DATA_BLOCK "DB240_Program10"   // DB240
{ S7_Optimized_Access := 'FALSE' }
AUTHOR : Robopac
VERSION : 0.0
// stored: AutoNumber false, IsOnlyStoredInLoadMemory false, IsWriteProtectedInAS false
   VAR RETAIN
      Program10 { S7_SetPoint := 'True'} : "DatiProgramma";
   END_VAR
BEGIN
   Program10.Wrapping := TRUE;
   Program10.TopLenght := 500;
   Program10.TopRelease := 0;
   Program10.TopDown := 0;
   Program10.Top := 4;
   Program10.PressurePTime := 0;
   Program10.LifterTime := 0;
   Program10.RevOverContrast := 1;
   Program10.RopeEndCycle := 16#02;
   Program10.Spare4 := 16#01;
   Program10.RopeTime := 1500;
   Program10.RevOverClamp := 1;
   Program10.FilmForceFinalRev := 10;
   Program10.FilmPrestretchFinalRev := 100;
   Program10.ArmSpeed := 100;
   Program10.CarriageDown4Top := 500;
   Program10.TopDownTime := 1500;
   Program10.LapsUnderTop := 0;
   Program10.Spare6 := 0;
   Program10.Spare7 := 0;
   Program10.Spare8 := 0;
   Program10.Spare9 := 0;
   Program10.Spare10 := 0;
   Program10.Spare11 := 0;
   Program10.Spare12 := 0;
   Program10.Overlap0_1 := 0;
   Program10.Height1 := 130;
   Program10.Landmark1 := FALSE;
   Program10.Lifter1 := FALSE;
   Program10.SpareBit1H1 := FALSE;
   Program10.Airblower1 := TRUE;
   Program10.NextStep1 := TRUE;
   Program10.PressureP1 := TRUE;
   Program10.SpareByte2H1 := 16#00;
   Program10.Revolution1 := 1;
   Program10.RopeUnit1_1 := 16#01;
   Program10.RopeUnit1_2 := 16#01;
   Program10.FilmForce1 := 5;
   Program10.FilmPrestretch1 := 200;
   Program10.Spare3H1 := 0;
   Program10.Spare49 := 0;
   Program10.Spare50 := 0;
   Program10.Spare51 := 0;
   Program10.Spare52 := 0;
   Program10.Spare53 := 0;
   Program10.Overlap1_2 := 0;
   Program10.Height2 := 50;
   Program10.Landmark2 := FALSE;
   Program10.Lifter2 := FALSE;
   Program10.SpareBit1H2 := FALSE;
   Program10.Airblower2 := TRUE;
   Program10.NextStep2 := TRUE;
   Program10.PressureP2 := TRUE;
   Program10.SpareByte2H2 := 16#00;
   Program10.Revolution2 := 1;
   Program10.RopeUnit2_1 := 16#01;
   Program10.RopeUnit2_2 := 16#01;
   Program10.FilmForce2 := 20;
   Program10.FilmPrestretch2 := 200;
   Program10.Spare3H2 := 0;
   Program10.Spare54 := 0;
   Program10.Spare55 := 0;
   Program10.Spare56 := 0;
   Program10.Spare57 := 0;
   Program10.Spare58 := 0;
   Program10.Overlap2_3 := 100;
   Program10.Height3 := -50;
   Program10.Landmark3 := TRUE;
   Program10.Lifter3 := FALSE;
   Program10.SpareBit1H3 := FALSE;
   Program10.Airblower3 := TRUE;
   Program10.NextStep3 := TRUE;
   Program10.PressureP3 := TRUE;
   Program10.SpareByte2H3 := 16#00;
   Program10.Revolution3 := 2;
   Program10.RopeUnit3_1 := 16#01;
   Program10.RopeUnit3_2 := 16#01;
   Program10.FilmForce3 := 30;
   Program10.FilmPrestretch3 := 200;
   Program10.Spare3H3 := 0;
   Program10.Spare59 := 0;
   Program10.Spare60 := 0;
   Program10.Spare61 := 380;
   Program10.Spare62 := 2800;
   Program10.Spare63 := 0;
   Program10.Overlap3_4 := 100;
   Program10.Height4 := 100;
   Program10.Landmark4 := FALSE;
   Program10.Lifter4 := FALSE;
   Program10.SpareBit1H4 := FALSE;
   Program10.Airblower4 := TRUE;
   Program10.NextStep4 := TRUE;
   Program10.PressureP4 := TRUE;
   Program10.SpareByte2H4 := 16#00;
   Program10.Revolution4 := 3;
   Program10.RopeUnit4_1 := 16#02;
   Program10.RopeUnit4_2 := 16#02;
   Program10.FilmForce4 := 30;
   Program10.FilmPrestretch4 := 200;
   Program10.Spare3H4 := 0;
   Program10.Spare64 := 0;
   Program10.Spare65 := 0;
   Program10.Spare66 := 0;
   Program10.Spare67 := 0;
   Program10.Spare68 := 0;
   Program10.Overlap4_5 := 0;
   Program10.Height5 := 50;
   Program10.Landmark5 := FALSE;
   Program10.Lifter5 := FALSE;
   Program10.SpareBit1H5 := FALSE;
   Program10.Airblower5 := TRUE;
   Program10.NextStep5 := FALSE;
   Program10.PressureP5 := FALSE;
   Program10.SpareByte2H5 := 16#00;
   Program10.Revolution5 := 1;
   Program10.RopeUnit5_1 := 16#01;
   Program10.RopeUnit5_2 := 16#01;
   Program10.FilmForce5 := 30;
   Program10.FilmPrestretch5 := 200;
   Program10.Spare3H5 := 0;
   Program10.Spare69 := 0;
   Program10.Spare70 := 0;
   Program10.Spare71 := 0;
   Program10.Spare72 := 0;
   Program10.Spare73 := 0;
   Program10.Overlap5_6 := 100;
   Program10.Height6 := 50;
   Program10.Landmark6 := FALSE;
   Program10.Lifter6 := FALSE;
   Program10.SpareBit1H6 := FALSE;
   Program10.Airblower6 := TRUE;
   Program10.NextStep6 := FALSE;
   Program10.PressureP6 := FALSE;
   Program10.SpareByte2H6 := 16#00;
   Program10.Revolution6 := 2;
   Program10.RopeUnit6_1 := 16#02;
   Program10.RopeUnit6_2 := 16#01;
   Program10.FilmForce6 := 20;
   Program10.FilmPrestretch6 := 200;
   Program10.Spare3H6 := 0;
   Program10.Spare74 := 0;
   Program10.Spare75 := 0;
   Program10.Spare76 := 0;
   Program10.Spare77 := 0;
   Program10.Spare78 := 0;
   Program10.Overlap6_7 := 0;
   Program10.Height7 := 0;
   Program10.Landmark7 := FALSE;
   Program10.Lifter7 := FALSE;
   Program10.SpareBit1H7 := FALSE;
   Program10.Airblower7 := FALSE;
   Program10.NextStep7 := TRUE;
   Program10.PressureP7 := FALSE;
   Program10.SpareByte2H7 := 16#00;
   Program10.Revolution7 := 1;
   Program10.RopeUnit7_1 := 16#01;
   Program10.RopeUnit7_2 := 16#01;
   Program10.FilmForce7 := 0;
   Program10.FilmPrestretch7 := 100;
   Program10.Spare3H7 := 0;
   Program10.Spare79 := 0;
   Program10.Spare80 := 0;
   Program10.Spare81 := 0;
   Program10.Spare82 := 0;
   Program10.Spare83 := 0;
   Program10.Overlap7_8 := 0;
   Program10.Height8 := 0;
   Program10.Landmark8 := FALSE;
   Program10.Lifter8 := FALSE;
   Program10.SpareBit1H8 := FALSE;
   Program10.Airblower8 := FALSE;
   Program10.NextStep8 := TRUE;
   Program10.PressureP8 := FALSE;
   Program10.SpareByte2H8 := 16#00;
   Program10.Revolution8 := 1;
   Program10.RopeUnit8_1 := 16#01;
   Program10.RopeUnit8_2 := 16#01;
   Program10.FilmForce8 := 0;
   Program10.FilmPrestretch8 := 100;
   Program10.Spare3H8 := 0;
   Program10.Spare84 := 0;
   Program10.Spare85 := 0;
   Program10.Spare86 := 0;
   Program10.Spare87 := 0;
   Program10.Spare88 := 0;
   Program10.Overlap8_9 := 0;
   Program10.Height9 := 0;
   Program10.Landmark9 := FALSE;
   Program10.Lifter9 := FALSE;
   Program10.SpareBit1H9 := FALSE;
   Program10.Airblower9 := FALSE;
   Program10.NextStep9 := TRUE;
   Program10.PressureP9 := FALSE;
   Program10.SpareByte2H9 := 16#00;
   Program10.Revolution9 := 1;
   Program10.RopeUnit9_1 := 16#01;
   Program10.RopeUnit9_2 := 16#01;
   Program10.FilmForce9 := 0;
   Program10.FilmPrestretch9 := 100;
   Program10.Spare3H9 := 0;
   Program10.Spare89 := 0;
   Program10.Spare90 := 0;
   Program10.Spare91 := 0;
   Program10.Spare92 := 0;
   Program10.Spare93 := 0;
   Program10.Overlap9_10 := 0;
   Program10.Height10 := 0;
   Program10.Landmark10 := FALSE;
   Program10.Lifter10 := FALSE;
   Program10.SpareBit1H10 := FALSE;
   Program10.Airblower10 := FALSE;
   Program10.NextStep10 := FALSE;
   Program10.PressureP10 := FALSE;
   Program10.SpareByte2H10 := 16#00;
   Program10.Revolution10 := 1;
   Program10.RopeUnit10_1 := 16#01;
   Program10.RopeUnit10_2 := 16#01;
   Program10.FilmForce10 := 0;
   Program10.FilmPrestretch10 := 100;
   Program10.Spare3H10 := 0;
   Program10.Spare94 := 0;
   Program10.Spare95 := 0;
   Program10.Spare96 := 0;
   Program10.Spare97 := 0;
   Program10.Spare98 := 0;
   Program10.Overlap10_11 := 0;
   Program10.Height11 := 0;
   Program10.Landmark11 := FALSE;
   Program10.Lifter11 := FALSE;
   Program10.SpareBit1H11 := FALSE;
   Program10.Airblower11 := FALSE;
   Program10.NextStep11 := TRUE;
   Program10.PressureP11 := FALSE;
   Program10.SpareByte2H11 := 16#00;
   Program10.Revolution11 := 1;
   Program10.RopeUnit11_1 := 16#01;
   Program10.RopeUnit11_2 := 16#01;
   Program10.FilmForce11 := 0;
   Program10.FilmPrestretch11 := 100;
   Program10.Spare3H11 := 0;
   Program10.Spare99 := 0;
   Program10.Spare100 := 0;
   Program10.Spare101 := 0;
   Program10.Spare102 := 0;
   Program10.Spare103 := 0;
   Program10.Overlap11_12 := 0;
   Program10.Height12 := 0;
   Program10.Landmark12 := FALSE;
   Program10.Lifter12 := FALSE;
   Program10.SpareBit1H12 := FALSE;
   Program10.Airblower12 := FALSE;
   Program10.NextStep12 := FALSE;
   Program10.PressureP12 := FALSE;
   Program10.SpareByte2H12 := 16#00;
   Program10.Revolution12 := 1;
   Program10.RopeUnit12_1 := 16#01;
   Program10.RopeUnit12_2 := 16#01;
   Program10.FilmForce12 := 0;
   Program10.FilmPrestretch12 := 100;
   Program10.Spare3H12 := 0;
   Program10.Spare104 := 0;
   Program10.Spare105 := 0;
   Program10.Spare106 := 0;
   Program10.Spare107 := 0;
   Program10.Spare108 := 0;
END_DATA_BLOCK

DATA_BLOCK "DB243_Program7"   // DB243
{ S7_Optimized_Access := 'FALSE' }
AUTHOR : Robopac
VERSION : 0.0
// stored: AutoNumber false, IsOnlyStoredInLoadMemory false, IsWriteProtectedInAS false
   VAR RETAIN
      Program7 { S7_SetPoint := 'True'} : "DatiProgramma";
   END_VAR
BEGIN
   Program7.Wrapping := TRUE;
   Program7.TopLenght := 500;
   Program7.TopRelease := 0;
   Program7.TopDown := 0;
   Program7.Top := 4;
   Program7.PressurePTime := 0;
   Program7.LifterTime := 0;
   Program7.RevOverContrast := 1;
   Program7.RopeEndCycle := 16#01;
   Program7.Spare4 := 16#01;
   Program7.RopeTime := 1500;
   Program7.RevOverClamp := 1;
   Program7.FilmForceFinalRev := 15;
   Program7.FilmPrestretchFinalRev := 100;
   Program7.ArmSpeed := 100;
   Program7.CarriageDown4Top := 500;
   Program7.TopDownTime := 1500;
   Program7.LapsUnderTop := 0;
   Program7.Spare6 := 0;
   Program7.Spare7 := 0;
   Program7.Spare8 := 0;
   Program7.Spare9 := 0;
   Program7.Spare10 := 0;
   Program7.Spare11 := 0;
   Program7.Spare12 := 0;
   Program7.Overlap0_1 := 0;
   Program7.Height1 := 15;
   Program7.Landmark1 := FALSE;
   Program7.Lifter1 := FALSE;
   Program7.SpareBit1H1 := FALSE;
   Program7.Airblower1 := TRUE;
   Program7.NextStep1 := TRUE;
   Program7.PressureP1 := TRUE;
   Program7.SpareByte2H1 := 16#00;
   Program7.Revolution1 := 0;
   Program7.RopeUnit1_1 := 16#02;
   Program7.RopeUnit1_2 := 16#01;
   Program7.FilmForce1 := 5;
   Program7.FilmPrestretch1 := 200;
   Program7.Spare3H1 := 0;
   Program7.Spare49 := 0;
   Program7.Spare50 := 0;
   Program7.Spare51 := 0;
   Program7.Spare52 := 0;
   Program7.Spare53 := 0;
   Program7.Overlap1_2 := 0;
   Program7.Height2 := 80;
   Program7.Landmark2 := FALSE;
   Program7.Lifter2 := FALSE;
   Program7.SpareBit1H2 := FALSE;
   Program7.Airblower2 := TRUE;
   Program7.NextStep2 := TRUE;
   Program7.PressureP2 := TRUE;
   Program7.SpareByte2H2 := 16#00;
   Program7.Revolution2 := 1;
   Program7.RopeUnit2_1 := 16#01;
   Program7.RopeUnit2_2 := 16#01;
   Program7.FilmForce2 := 15;
   Program7.FilmPrestretch2 := 200;
   Program7.Spare3H2 := 0;
   Program7.Spare54 := 0;
   Program7.Spare55 := 0;
   Program7.Spare56 := 0;
   Program7.Spare57 := 0;
   Program7.Spare58 := 0;
   Program7.Overlap2_3 := 0;
   Program7.Height3 := 120;
   Program7.Landmark3 := FALSE;
   Program7.Lifter3 := FALSE;
   Program7.SpareBit1H3 := FALSE;
   Program7.Airblower3 := TRUE;
   Program7.NextStep3 := TRUE;
   Program7.PressureP3 := TRUE;
   Program7.SpareByte2H3 := 16#00;
   Program7.Revolution3 := 1;
   Program7.RopeUnit3_1 := 16#01;
   Program7.RopeUnit3_2 := 16#01;
   Program7.FilmForce3 := 25;
   Program7.FilmPrestretch3 := 200;
   Program7.Spare3H3 := 0;
   Program7.Spare59 := 0;
   Program7.Spare60 := 0;
   Program7.Spare61 := 380;
   Program7.Spare62 := 2800;
   Program7.Spare63 := 0;
   Program7.Overlap3_4 := 0;
   Program7.Height4 := -100;
   Program7.Landmark4 := TRUE;
   Program7.Lifter4 := FALSE;
   Program7.SpareBit1H4 := FALSE;
   Program7.Airblower4 := FALSE;
   Program7.NextStep4 := TRUE;
   Program7.PressureP4 := TRUE;
   Program7.SpareByte2H4 := 16#00;
   Program7.Revolution4 := 1;
   Program7.RopeUnit4_1 := 16#01;
   Program7.RopeUnit4_2 := 16#01;
   Program7.FilmForce4 := 20;
   Program7.FilmPrestretch4 := 200;
   Program7.Spare3H4 := 0;
   Program7.Spare64 := 0;
   Program7.Spare65 := 0;
   Program7.Spare66 := 0;
   Program7.Spare67 := 0;
   Program7.Spare68 := 0;
   Program7.Overlap4_5 := 300;
   Program7.Height5 := 120;
   Program7.Landmark5 := FALSE;
   Program7.Lifter5 := FALSE;
   Program7.SpareBit1H5 := FALSE;
   Program7.Airblower5 := TRUE;
   Program7.NextStep5 := TRUE;
   Program7.PressureP5 := FALSE;
   Program7.SpareByte2H5 := 16#00;
   Program7.Revolution5 := 2;
   Program7.RopeUnit5_1 := 16#02;
   Program7.RopeUnit5_2 := 16#02;
   Program7.FilmForce5 := 15;
   Program7.FilmPrestretch5 := 200;
   Program7.Spare3H5 := 0;
   Program7.Spare69 := 0;
   Program7.Spare70 := 0;
   Program7.Spare71 := 0;
   Program7.Spare72 := 0;
   Program7.Spare73 := 0;
   Program7.Overlap5_6 := 300;
   Program7.Height6 := 85;
   Program7.Landmark6 := FALSE;
   Program7.Lifter6 := FALSE;
   Program7.SpareBit1H6 := FALSE;
   Program7.Airblower6 := TRUE;
   Program7.NextStep6 := FALSE;
   Program7.PressureP6 := FALSE;
   Program7.SpareByte2H6 := 16#00;
   Program7.Revolution6 := 1;
   Program7.RopeUnit6_1 := 16#01;
   Program7.RopeUnit6_2 := 16#01;
   Program7.FilmForce6 := 20;
   Program7.FilmPrestretch6 := 200;
   Program7.Spare3H6 := 0;
   Program7.Spare74 := 0;
   Program7.Spare75 := 0;
   Program7.Spare76 := 0;
   Program7.Spare77 := 0;
   Program7.Spare78 := 0;
   Program7.Overlap6_7 := 0;
   Program7.Height7 := 0;
   Program7.Landmark7 := FALSE;
   Program7.Lifter7 := FALSE;
   Program7.SpareBit1H7 := FALSE;
   Program7.Airblower7 := FALSE;
   Program7.NextStep7 := TRUE;
   Program7.PressureP7 := FALSE;
   Program7.SpareByte2H7 := 16#00;
   Program7.Revolution7 := 1;
   Program7.RopeUnit7_1 := 16#01;
   Program7.RopeUnit7_2 := 16#01;
   Program7.FilmForce7 := 0;
   Program7.FilmPrestretch7 := 100;
   Program7.Spare3H7 := 0;
   Program7.Spare79 := 0;
   Program7.Spare80 := 0;
   Program7.Spare81 := 0;
   Program7.Spare82 := 0;
   Program7.Spare83 := 0;
   Program7.Overlap7_8 := 0;
   Program7.Height8 := 0;
   Program7.Landmark8 := FALSE;
   Program7.Lifter8 := FALSE;
   Program7.SpareBit1H8 := FALSE;
   Program7.Airblower8 := FALSE;
   Program7.NextStep8 := TRUE;
   Program7.PressureP8 := FALSE;
   Program7.SpareByte2H8 := 16#00;
   Program7.Revolution8 := 1;
   Program7.RopeUnit8_1 := 16#01;
   Program7.RopeUnit8_2 := 16#01;
   Program7.FilmForce8 := 0;
   Program7.FilmPrestretch8 := 100;
   Program7.Spare3H8 := 0;
   Program7.Spare84 := 0;
   Program7.Spare85 := 0;
   Program7.Spare86 := 0;
   Program7.Spare87 := 0;
   Program7.Spare88 := 0;
   Program7.Overlap8_9 := 0;
   Program7.Height9 := 0;
   Program7.Landmark9 := FALSE;
   Program7.Lifter9 := FALSE;
   Program7.SpareBit1H9 := FALSE;
   Program7.Airblower9 := FALSE;
   Program7.NextStep9 := TRUE;
   Program7.PressureP9 := FALSE;
   Program7.SpareByte2H9 := 16#00;
   Program7.Revolution9 := 1;
   Program7.RopeUnit9_1 := 16#01;
   Program7.RopeUnit9_2 := 16#01;
   Program7.FilmForce9 := 0;
   Program7.FilmPrestretch9 := 100;
   Program7.Spare3H9 := 0;
   Program7.Spare89 := 0;
   Program7.Spare90 := 0;
   Program7.Spare91 := 0;
   Program7.Spare92 := 0;
   Program7.Spare93 := 0;
   Program7.Overlap9_10 := 0;
   Program7.Height10 := 0;
   Program7.Landmark10 := FALSE;
   Program7.Lifter10 := FALSE;
   Program7.SpareBit1H10 := FALSE;
   Program7.Airblower10 := FALSE;
   Program7.NextStep10 := FALSE;
   Program7.PressureP10 := FALSE;
   Program7.SpareByte2H10 := 16#00;
   Program7.Revolution10 := 1;
   Program7.RopeUnit10_1 := 16#01;
   Program7.RopeUnit10_2 := 16#01;
   Program7.FilmForce10 := 0;
   Program7.FilmPrestretch10 := 100;
   Program7.Spare3H10 := 0;
   Program7.Spare94 := 0;
   Program7.Spare95 := 0;
   Program7.Spare96 := 0;
   Program7.Spare97 := 0;
   Program7.Spare98 := 0;
   Program7.Overlap10_11 := 0;
   Program7.Height11 := 0;
   Program7.Landmark11 := FALSE;
   Program7.Lifter11 := FALSE;
   Program7.SpareBit1H11 := FALSE;
   Program7.Airblower11 := FALSE;
   Program7.NextStep11 := TRUE;
   Program7.PressureP11 := FALSE;
   Program7.SpareByte2H11 := 16#00;
   Program7.Revolution11 := 1;
   Program7.RopeUnit11_1 := 16#01;
   Program7.RopeUnit11_2 := 16#01;
   Program7.FilmForce11 := 0;
   Program7.FilmPrestretch11 := 100;
   Program7.Spare3H11 := 0;
   Program7.Spare99 := 0;
   Program7.Spare100 := 0;
   Program7.Spare101 := 0;
   Program7.Spare102 := 0;
   Program7.Spare103 := 0;
   Program7.Overlap11_12 := 0;
   Program7.Height12 := 0;
   Program7.Landmark12 := FALSE;
   Program7.Lifter12 := FALSE;
   Program7.SpareBit1H12 := FALSE;
   Program7.Airblower12 := FALSE;
   Program7.NextStep12 := FALSE;
   Program7.PressureP12 := FALSE;
   Program7.SpareByte2H12 := 16#00;
   Program7.Revolution12 := 1;
   Program7.RopeUnit12_1 := 16#01;
   Program7.RopeUnit12_2 := 16#01;
   Program7.FilmForce12 := 0;
   Program7.FilmPrestretch12 := 100;
   Program7.Spare3H12 := 0;
   Program7.Spare104 := 0;
   Program7.Spare105 := 0;
   Program7.Spare106 := 0;
   Program7.Spare107 := 0;
   Program7.Spare108 := 0;
END_DATA_BLOCK

DATA_BLOCK "DB246_Program4"   // DB246
{ S7_Optimized_Access := 'FALSE' }
AUTHOR : Robopac
VERSION : 0.0
// stored: AutoNumber false, IsOnlyStoredInLoadMemory false, IsWriteProtectedInAS false
   VAR RETAIN
      Program4 { S7_SetPoint := 'True'} : "DatiProgramma";
   END_VAR
BEGIN
   Program4.Wrapping := TRUE;
   Program4.TopLenght := 500;
   Program4.TopRelease := 0;
   Program4.TopDown := 0;
   Program4.Top := 4;
   Program4.PressurePTime := 0;
   Program4.LifterTime := 0;
   Program4.RevOverContrast := 1;
   Program4.RopeEndCycle := 16#02;
   Program4.Spare4 := 16#01;
   Program4.RopeTime := 1500;
   Program4.RevOverClamp := 1;
   Program4.FilmForceFinalRev := 10;
   Program4.FilmPrestretchFinalRev := 100;
   Program4.ArmSpeed := 100;
   Program4.CarriageDown4Top := 500;
   Program4.TopDownTime := 1500;
   Program4.LapsUnderTop := 0;
   Program4.Spare6 := 0;
   Program4.Spare7 := 0;
   Program4.Spare8 := 0;
   Program4.Spare9 := 0;
   Program4.Spare10 := 0;
   Program4.Spare11 := 0;
   Program4.Spare12 := 0;
   Program4.Overlap0_1 := 0;
   Program4.Height1 := 130;
   Program4.Landmark1 := FALSE;
   Program4.Lifter1 := FALSE;
   Program4.SpareBit1H1 := FALSE;
   Program4.Airblower1 := TRUE;
   Program4.NextStep1 := TRUE;
   Program4.PressureP1 := TRUE;
   Program4.SpareByte2H1 := 16#00;
   Program4.Revolution1 := 1;
   Program4.RopeUnit1_1 := 16#01;
   Program4.RopeUnit1_2 := 16#01;
   Program4.FilmForce1 := 5;
   Program4.FilmPrestretch1 := 200;
   Program4.Spare3H1 := 0;
   Program4.Spare49 := 0;
   Program4.Spare50 := 0;
   Program4.Spare51 := 0;
   Program4.Spare52 := 0;
   Program4.Spare53 := 0;
   Program4.Overlap1_2 := 0;
   Program4.Height2 := 50;
   Program4.Landmark2 := FALSE;
   Program4.Lifter2 := FALSE;
   Program4.SpareBit1H2 := FALSE;
   Program4.Airblower2 := TRUE;
   Program4.NextStep2 := TRUE;
   Program4.PressureP2 := TRUE;
   Program4.SpareByte2H2 := 16#00;
   Program4.Revolution2 := 1;
   Program4.RopeUnit2_1 := 16#01;
   Program4.RopeUnit2_2 := 16#01;
   Program4.FilmForce2 := 20;
   Program4.FilmPrestretch2 := 200;
   Program4.Spare3H2 := 0;
   Program4.Spare54 := 0;
   Program4.Spare55 := 0;
   Program4.Spare56 := 0;
   Program4.Spare57 := 0;
   Program4.Spare58 := 0;
   Program4.Overlap2_3 := 100;
   Program4.Height3 := -50;
   Program4.Landmark3 := TRUE;
   Program4.Lifter3 := FALSE;
   Program4.SpareBit1H3 := FALSE;
   Program4.Airblower3 := TRUE;
   Program4.NextStep3 := TRUE;
   Program4.PressureP3 := TRUE;
   Program4.SpareByte2H3 := 16#00;
   Program4.Revolution3 := 2;
   Program4.RopeUnit3_1 := 16#01;
   Program4.RopeUnit3_2 := 16#01;
   Program4.FilmForce3 := 30;
   Program4.FilmPrestretch3 := 200;
   Program4.Spare3H3 := 0;
   Program4.Spare59 := 0;
   Program4.Spare60 := 0;
   Program4.Spare61 := 380;
   Program4.Spare62 := 2800;
   Program4.Spare63 := 0;
   Program4.Overlap3_4 := 100;
   Program4.Height4 := 100;
   Program4.Landmark4 := FALSE;
   Program4.Lifter4 := FALSE;
   Program4.SpareBit1H4 := FALSE;
   Program4.Airblower4 := TRUE;
   Program4.NextStep4 := TRUE;
   Program4.PressureP4 := TRUE;
   Program4.SpareByte2H4 := 16#00;
   Program4.Revolution4 := 3;
   Program4.RopeUnit4_1 := 16#02;
   Program4.RopeUnit4_2 := 16#02;
   Program4.FilmForce4 := 30;
   Program4.FilmPrestretch4 := 200;
   Program4.Spare3H4 := 0;
   Program4.Spare64 := 0;
   Program4.Spare65 := 0;
   Program4.Spare66 := 0;
   Program4.Spare67 := 0;
   Program4.Spare68 := 0;
   Program4.Overlap4_5 := 0;
   Program4.Height5 := 50;
   Program4.Landmark5 := FALSE;
   Program4.Lifter5 := FALSE;
   Program4.SpareBit1H5 := FALSE;
   Program4.Airblower5 := TRUE;
   Program4.NextStep5 := FALSE;
   Program4.PressureP5 := FALSE;
   Program4.SpareByte2H5 := 16#00;
   Program4.Revolution5 := 1;
   Program4.RopeUnit5_1 := 16#01;
   Program4.RopeUnit5_2 := 16#01;
   Program4.FilmForce5 := 30;
   Program4.FilmPrestretch5 := 200;
   Program4.Spare3H5 := 0;
   Program4.Spare69 := 0;
   Program4.Spare70 := 0;
   Program4.Spare71 := 0;
   Program4.Spare72 := 0;
   Program4.Spare73 := 0;
   Program4.Overlap5_6 := 100;
   Program4.Height6 := 50;
   Program4.Landmark6 := FALSE;
   Program4.Lifter6 := FALSE;
   Program4.SpareBit1H6 := FALSE;
   Program4.Airblower6 := TRUE;
   Program4.NextStep6 := FALSE;
   Program4.PressureP6 := FALSE;
   Program4.SpareByte2H6 := 16#00;
   Program4.Revolution6 := 2;
   Program4.RopeUnit6_1 := 16#02;
   Program4.RopeUnit6_2 := 16#01;
   Program4.FilmForce6 := 20;
   Program4.FilmPrestretch6 := 200;
   Program4.Spare3H6 := 0;
   Program4.Spare74 := 0;
   Program4.Spare75 := 0;
   Program4.Spare76 := 0;
   Program4.Spare77 := 0;
   Program4.Spare78 := 0;
   Program4.Overlap6_7 := 0;
   Program4.Height7 := 0;
   Program4.Landmark7 := FALSE;
   Program4.Lifter7 := FALSE;
   Program4.SpareBit1H7 := FALSE;
   Program4.Airblower7 := FALSE;
   Program4.NextStep7 := TRUE;
   Program4.PressureP7 := FALSE;
   Program4.SpareByte2H7 := 16#00;
   Program4.Revolution7 := 1;
   Program4.RopeUnit7_1 := 16#01;
   Program4.RopeUnit7_2 := 16#01;
   Program4.FilmForce7 := 0;
   Program4.FilmPrestretch7 := 100;
   Program4.Spare3H7 := 0;
   Program4.Spare79 := 0;
   Program4.Spare80 := 0;
   Program4.Spare81 := 0;
   Program4.Spare82 := 0;
   Program4.Spare83 := 0;
   Program4.Overlap7_8 := 0;
   Program4.Height8 := 0;
   Program4.Landmark8 := FALSE;
   Program4.Lifter8 := FALSE;
   Program4.SpareBit1H8 := FALSE;
   Program4.Airblower8 := FALSE;
   Program4.NextStep8 := TRUE;
   Program4.PressureP8 := FALSE;
   Program4.SpareByte2H8 := 16#00;
   Program4.Revolution8 := 1;
   Program4.RopeUnit8_1 := 16#01;
   Program4.RopeUnit8_2 := 16#01;
   Program4.FilmForce8 := 0;
   Program4.FilmPrestretch8 := 100;
   Program4.Spare3H8 := 0;
   Program4.Spare84 := 0;
   Program4.Spare85 := 0;
   Program4.Spare86 := 0;
   Program4.Spare87 := 0;
   Program4.Spare88 := 0;
   Program4.Overlap8_9 := 0;
   Program4.Height9 := 0;
   Program4.Landmark9 := FALSE;
   Program4.Lifter9 := FALSE;
   Program4.SpareBit1H9 := FALSE;
   Program4.Airblower9 := FALSE;
   Program4.NextStep9 := TRUE;
   Program4.PressureP9 := FALSE;
   Program4.SpareByte2H9 := 16#00;
   Program4.Revolution9 := 1;
   Program4.RopeUnit9_1 := 16#01;
   Program4.RopeUnit9_2 := 16#01;
   Program4.FilmForce9 := 0;
   Program4.FilmPrestretch9 := 100;
   Program4.Spare3H9 := 0;
   Program4.Spare89 := 0;
   Program4.Spare90 := 0;
   Program4.Spare91 := 0;
   Program4.Spare92 := 0;
   Program4.Spare93 := 0;
   Program4.Overlap9_10 := 0;
   Program4.Height10 := 0;
   Program4.Landmark10 := FALSE;
   Program4.Lifter10 := FALSE;
   Program4.SpareBit1H10 := FALSE;
   Program4.Airblower10 := FALSE;
   Program4.NextStep10 := FALSE;
   Program4.PressureP10 := FALSE;
   Program4.SpareByte2H10 := 16#00;
   Program4.Revolution10 := 1;
   Program4.RopeUnit10_1 := 16#01;
   Program4.RopeUnit10_2 := 16#01;
   Program4.FilmForce10 := 0;
   Program4.FilmPrestretch10 := 100;
   Program4.Spare3H10 := 0;
   Program4.Spare94 := 0;
   Program4.Spare95 := 0;
   Program4.Spare96 := 0;
   Program4.Spare97 := 0;
   Program4.Spare98 := 0;
   Program4.Overlap10_11 := 0;
   Program4.Height11 := 0;
   Program4.Landmark11 := FALSE;
   Program4.Lifter11 := FALSE;
   Program4.SpareBit1H11 := FALSE;
   Program4.Airblower11 := FALSE;
   Program4.NextStep11 := TRUE;
   Program4.PressureP11 := FALSE;
   Program4.SpareByte2H11 := 16#00;
   Program4.Revolution11 := 1;
   Program4.RopeUnit11_1 := 16#01;
   Program4.RopeUnit11_2 := 16#01;
   Program4.FilmForce11 := 0;
   Program4.FilmPrestretch11 := 100;
   Program4.Spare3H11 := 0;
   Program4.Spare99 := 0;
   Program4.Spare100 := 0;
   Program4.Spare101 := 0;
   Program4.Spare102 := 0;
   Program4.Spare103 := 0;
   Program4.Overlap11_12 := 0;
   Program4.Height12 := 0;
   Program4.Landmark12 := FALSE;
   Program4.Lifter12 := FALSE;
   Program4.SpareBit1H12 := FALSE;
   Program4.Airblower12 := FALSE;
   Program4.NextStep12 := FALSE;
   Program4.PressureP12 := FALSE;
   Program4.SpareByte2H12 := 16#00;
   Program4.Revolution12 := 1;
   Program4.RopeUnit12_1 := 16#01;
   Program4.RopeUnit12_2 := 16#01;
   Program4.FilmForce12 := 0;
   Program4.FilmPrestretch12 := 100;
   Program4.Spare3H12 := 0;
   Program4.Spare104 := 0;
   Program4.Spare105 := 0;
   Program4.Spare106 := 0;
   Program4.Spare107 := 0;
   Program4.Spare108 := 0;
END_DATA_BLOCK

DATA_BLOCK "DB249_Program1"   // DB249
{ S7_Optimized_Access := 'FALSE' }
AUTHOR : Robopac
VERSION : 0.0
// stored: AutoNumber false, IsOnlyStoredInLoadMemory false, IsWriteProtectedInAS false
   VAR RETAIN
      Program1 { S7_SetPoint := 'True'} : "DatiProgramma";
   END_VAR
BEGIN
   Program1.Wrapping := TRUE;
   Program1.TopLenght := 500;
   Program1.TopRelease := 0;
   Program1.TopDown := 0;
   Program1.Top := 4;
   Program1.PressurePTime := 0;
   Program1.LifterTime := 0;
   Program1.RevOverContrast := 1;
   Program1.RopeEndCycle := 16#02;
   Program1.Spare4 := 16#01;
   Program1.RopeTime := 1500;
   Program1.RevOverClamp := 1;
   Program1.FilmForceFinalRev := 25;
   Program1.FilmPrestretchFinalRev := 100;
   Program1.ArmSpeed := 87;
   Program1.CarriageDown4Top := 500;
   Program1.TopDownTime := 1500;
   Program1.LapsUnderTop := 0;
   Program1.Spare6 := 0;
   Program1.Spare7 := 0;
   Program1.Spare8 := 0;
   Program1.Spare9 := 0;
   Program1.Spare10 := 0;
   Program1.Spare11 := 0;
   Program1.Spare12 := 0;
   Program1.Overlap0_1 := 0;
   Program1.Height1 := 120;
   Program1.Landmark1 := FALSE;
   Program1.Lifter1 := FALSE;
   Program1.SpareBit1H1 := FALSE;
   Program1.Airblower1 := TRUE;
   Program1.NextStep1 := TRUE;
   Program1.PressureP1 := TRUE;
   Program1.SpareByte2H1 := 16#00;
   Program1.Revolution1 := 1;
   Program1.RopeUnit1_1 := 16#03;
   Program1.RopeUnit1_2 := 16#01;
   Program1.FilmForce1 := 5;
   Program1.FilmPrestretch1 := 200;
   Program1.Spare3H1 := 0;
   Program1.Spare49 := 0;
   Program1.Spare50 := 0;
   Program1.Spare51 := 0;
   Program1.Spare52 := 0;
   Program1.Spare53 := 0;
   Program1.Overlap1_2 := 0;
   Program1.Height2 := 85;
   Program1.Landmark2 := FALSE;
   Program1.Lifter2 := FALSE;
   Program1.SpareBit1H2 := FALSE;
   Program1.Airblower2 := TRUE;
   Program1.NextStep2 := TRUE;
   Program1.PressureP2 := TRUE;
   Program1.SpareByte2H2 := 16#00;
   Program1.Revolution2 := 3;
   Program1.RopeUnit2_1 := 16#01;
   Program1.RopeUnit2_2 := 16#01;
   Program1.FilmForce2 := 15;
   Program1.FilmPrestretch2 := 200;
   Program1.Spare3H2 := 0;
   Program1.Spare54 := 0;
   Program1.Spare55 := 0;
   Program1.Spare56 := 0;
   Program1.Spare57 := 0;
   Program1.Spare58 := 0;
   Program1.Overlap2_3 := 300;
   Program1.Height3 := 110;
   Program1.Landmark3 := FALSE;
   Program1.Lifter3 := FALSE;
   Program1.SpareBit1H3 := FALSE;
   Program1.Airblower3 := TRUE;
   Program1.NextStep3 := TRUE;
   Program1.PressureP3 := TRUE;
   Program1.SpareByte2H3 := 16#00;
   Program1.Revolution3 := 2;
   Program1.RopeUnit3_1 := 16#03;
   Program1.RopeUnit3_2 := 16#03;
   Program1.FilmForce3 := 20;
   Program1.FilmPrestretch3 := 200;
   Program1.Spare3H3 := 0;
   Program1.Spare59 := 0;
   Program1.Spare60 := 0;
   Program1.Spare61 := 380;
   Program1.Spare62 := 2800;
   Program1.Spare63 := 0;
   Program1.Overlap3_4 := 100;
   Program1.Height4 := -100;
   Program1.Landmark4 := TRUE;
   Program1.Lifter4 := FALSE;
   Program1.SpareBit1H4 := FALSE;
   Program1.Airblower4 := FALSE;
   Program1.NextStep4 := TRUE;
   Program1.PressureP4 := TRUE;
   Program1.SpareByte2H4 := 16#00;
   Program1.Revolution4 := 1;
   Program1.RopeUnit4_1 := 16#01;
   Program1.RopeUnit4_2 := 16#01;
   Program1.FilmForce4 := 18;
   Program1.FilmPrestretch4 := 200;
   Program1.Spare3H4 := 0;
   Program1.Spare64 := 0;
   Program1.Spare65 := 0;
   Program1.Spare66 := 0;
   Program1.Spare67 := 0;
   Program1.Spare68 := 0;
   Program1.Overlap4_5 := 100;
   Program1.Height5 := 60;
   Program1.Landmark5 := FALSE;
   Program1.Lifter5 := FALSE;
   Program1.SpareBit1H5 := FALSE;
   Program1.Airblower5 := TRUE;
   Program1.NextStep5 := TRUE;
   Program1.PressureP5 := FALSE;
   Program1.SpareByte2H5 := 16#00;
   Program1.Revolution5 := 1;
   Program1.RopeUnit5_1 := 16#01;
   Program1.RopeUnit5_2 := 16#01;
   Program1.FilmForce5 := 25;
   Program1.FilmPrestretch5 := 200;
   Program1.Spare3H5 := 0;
   Program1.Spare69 := 0;
   Program1.Spare70 := 0;
   Program1.Spare71 := 0;
   Program1.Spare72 := 0;
   Program1.Spare73 := 0;
   Program1.Overlap5_6 := 100;
   Program1.Height6 := 40;
   Program1.Landmark6 := FALSE;
   Program1.Lifter6 := FALSE;
   Program1.SpareBit1H6 := FALSE;
   Program1.Airblower6 := TRUE;
   Program1.NextStep6 := FALSE;
   Program1.PressureP6 := FALSE;
   Program1.SpareByte2H6 := 16#00;
   Program1.Revolution6 := 1;
   Program1.RopeUnit6_1 := 16#01;
   Program1.RopeUnit6_2 := 16#01;
   Program1.FilmForce6 := 15;
   Program1.FilmPrestretch6 := 200;
   Program1.Spare3H6 := 0;
   Program1.Spare74 := 0;
   Program1.Spare75 := 0;
   Program1.Spare76 := 0;
   Program1.Spare77 := 0;
   Program1.Spare78 := 0;
   Program1.Overlap6_7 := 0;
   Program1.Height7 := 0;
   Program1.Landmark7 := FALSE;
   Program1.Lifter7 := FALSE;
   Program1.SpareBit1H7 := FALSE;
   Program1.Airblower7 := FALSE;
   Program1.NextStep7 := TRUE;
   Program1.PressureP7 := FALSE;
   Program1.SpareByte2H7 := 16#00;
   Program1.Revolution7 := 1;
   Program1.RopeUnit7_1 := 16#01;
   Program1.RopeUnit7_2 := 16#01;
   Program1.FilmForce7 := 0;
   Program1.FilmPrestretch7 := 100;
   Program1.Spare3H7 := 0;
   Program1.Spare79 := 0;
   Program1.Spare80 := 0;
   Program1.Spare81 := 0;
   Program1.Spare82 := 0;
   Program1.Spare83 := 0;
   Program1.Overlap7_8 := 0;
   Program1.Height8 := 0;
   Program1.Landmark8 := FALSE;
   Program1.Lifter8 := FALSE;
   Program1.SpareBit1H8 := FALSE;
   Program1.Airblower8 := FALSE;
   Program1.NextStep8 := TRUE;
   Program1.PressureP8 := FALSE;
   Program1.SpareByte2H8 := 16#00;
   Program1.Revolution8 := 1;
   Program1.RopeUnit8_1 := 16#01;
   Program1.RopeUnit8_2 := 16#01;
   Program1.FilmForce8 := 0;
   Program1.FilmPrestretch8 := 100;
   Program1.Spare3H8 := 0;
   Program1.Spare84 := 0;
   Program1.Spare85 := 0;
   Program1.Spare86 := 0;
   Program1.Spare87 := 0;
   Program1.Spare88 := 0;
   Program1.Overlap8_9 := 0;
   Program1.Height9 := 0;
   Program1.Landmark9 := FALSE;
   Program1.Lifter9 := FALSE;
   Program1.SpareBit1H9 := FALSE;
   Program1.Airblower9 := FALSE;
   Program1.NextStep9 := TRUE;
   Program1.PressureP9 := FALSE;
   Program1.SpareByte2H9 := 16#00;
   Program1.Revolution9 := 1;
   Program1.RopeUnit9_1 := 16#01;
   Program1.RopeUnit9_2 := 16#01;
   Program1.FilmForce9 := 0;
   Program1.FilmPrestretch9 := 100;
   Program1.Spare3H9 := 0;
   Program1.Spare89 := 0;
   Program1.Spare90 := 0;
   Program1.Spare91 := 0;
   Program1.Spare92 := 0;
   Program1.Spare93 := 0;
   Program1.Overlap9_10 := 0;
   Program1.Height10 := 0;
   Program1.Landmark10 := FALSE;
   Program1.Lifter10 := FALSE;
   Program1.SpareBit1H10 := FALSE;
   Program1.Airblower10 := FALSE;
   Program1.NextStep10 := FALSE;
   Program1.PressureP10 := FALSE;
   Program1.SpareByte2H10 := 16#00;
   Program1.Revolution10 := 1;
   Program1.RopeUnit10_1 := 16#01;
   Program1.RopeUnit10_2 := 16#01;
   Program1.FilmForce10 := 0;
   Program1.FilmPrestretch10 := 100;
   Program1.Spare3H10 := 0;
   Program1.Spare94 := 0;
   Program1.Spare95 := 0;
   Program1.Spare96 := 0;
   Program1.Spare97 := 0;
   Program1.Spare98 := 0;
   Program1.Overlap10_11 := 0;
   Program1.Height11 := 0;
   Program1.Landmark11 := FALSE;
   Program1.Lifter11 := FALSE;
   Program1.SpareBit1H11 := FALSE;
   Program1.Airblower11 := FALSE;
   Program1.NextStep11 := TRUE;
   Program1.PressureP11 := FALSE;
   Program1.SpareByte2H11 := 16#00;
   Program1.Revolution11 := 1;
   Program1.RopeUnit11_1 := 16#01;
   Program1.RopeUnit11_2 := 16#01;
   Program1.FilmForce11 := 0;
   Program1.FilmPrestretch11 := 100;
   Program1.Spare3H11 := 0;
   Program1.Spare99 := 0;
   Program1.Spare100 := 0;
   Program1.Spare101 := 0;
   Program1.Spare102 := 0;
   Program1.Spare103 := 0;
   Program1.Overlap11_12 := 0;
   Program1.Height12 := 0;
   Program1.Landmark12 := FALSE;
   Program1.Lifter12 := FALSE;
   Program1.SpareBit1H12 := FALSE;
   Program1.Airblower12 := FALSE;
   Program1.NextStep12 := FALSE;
   Program1.PressureP12 := FALSE;
   Program1.SpareByte2H12 := 16#00;
   Program1.Revolution12 := 1;
   Program1.RopeUnit12_1 := 16#01;
   Program1.RopeUnit12_2 := 16#01;
   Program1.FilmForce12 := 0;
   Program1.FilmPrestretch12 := 100;
   Program1.Spare3H12 := 0;
   Program1.Spare104 := 0;
   Program1.Spare105 := 0;
   Program1.Spare106 := 0;
   Program1.Spare107 := 0;
   Program1.Spare108 := 0;
END_DATA_BLOCK

DATA_BLOCK "DB250_ProgramData"   // DB250
{ S7_Optimized_Access := 'FALSE' }
AUTHOR : Robopac
VERSION : 0.0
// stored: AutoNumber false, IsOnlyStoredInLoadMemory false, IsWriteProtectedInAS false
   VAR RETAIN
      Program { S7_SetPoint := 'True'} : "DatiProgramma";
   END_VAR
BEGIN
   Program.Wrapping := TRUE;
   Program.TopLenght := 500;
   Program.TopRelease := 0;
   Program.TopDown := 0;
   Program.Top := 4;
   Program.PressurePTime := 0;
   Program.LifterTime := 0;
   Program.RevOverContrast := 1;
   Program.RopeEndCycle := 16#02;
   Program.Spare4 := 16#01;
   Program.RopeTime := 1500;
   Program.RevOverClamp := 1;
   Program.FilmForceFinalRev := 10;
   Program.FilmPrestretchFinalRev := 100;
   Program.ArmSpeed := 100;
   Program.CarriageDown4Top := 500;
   Program.TopDownTime := 1500;
   Program.LapsUnderTop := 0;
   Program.Spare6 := 0;
   Program.Spare7 := 0;
   Program.Spare8 := 0;
   Program.Spare9 := 0;
   Program.Spare10 := 0;
   Program.Spare11 := 0;
   Program.Spare12 := 0;
   Program.Overlap0_1 := 0;
   Program.Height1 := 130;
   Program.Landmark1 := FALSE;
   Program.Lifter1 := FALSE;
   Program.SpareBit1H1 := FALSE;
   Program.Airblower1 := TRUE;
   Program.NextStep1 := TRUE;
   Program.PressureP1 := TRUE;
   Program.SpareByte2H1 := 16#00;
   Program.Revolution1 := 1;
   Program.RopeUnit1_1 := 16#01;
   Program.RopeUnit1_2 := 16#01;
   Program.FilmForce1 := 5;
   Program.FilmPrestretch1 := 200;
   Program.Spare3H1 := 0;
   Program.Spare49 := 0;
   Program.Spare50 := 0;
   Program.Spare51 := 0;
   Program.Spare52 := 0;
   Program.Spare53 := 0;
   Program.Overlap1_2 := 0;
   Program.Height2 := 50;
   Program.Landmark2 := FALSE;
   Program.Lifter2 := FALSE;
   Program.SpareBit1H2 := FALSE;
   Program.Airblower2 := TRUE;
   Program.NextStep2 := TRUE;
   Program.PressureP2 := TRUE;
   Program.SpareByte2H2 := 16#00;
   Program.Revolution2 := 1;
   Program.RopeUnit2_1 := 16#01;
   Program.RopeUnit2_2 := 16#01;
   Program.FilmForce2 := 20;
   Program.FilmPrestretch2 := 200;
   Program.Spare3H2 := 0;
   Program.Spare54 := 0;
   Program.Spare55 := 0;
   Program.Spare56 := 0;
   Program.Spare57 := 0;
   Program.Spare58 := 0;
   Program.Overlap2_3 := 100;
   Program.Height3 := -50;
   Program.Landmark3 := TRUE;
   Program.Lifter3 := FALSE;
   Program.SpareBit1H3 := FALSE;
   Program.Airblower3 := TRUE;
   Program.NextStep3 := TRUE;
   Program.PressureP3 := TRUE;
   Program.SpareByte2H3 := 16#00;
   Program.Revolution3 := 2;
   Program.RopeUnit3_1 := 16#01;
   Program.RopeUnit3_2 := 16#01;
   Program.FilmForce3 := 30;
   Program.FilmPrestretch3 := 200;
   Program.Spare3H3 := 0;
   Program.Spare59 := 0;
   Program.Spare60 := 0;
   Program.Spare61 := 380;
   Program.Spare62 := 2800;
   Program.Spare63 := 0;
   Program.Overlap3_4 := 100;
   Program.Height4 := 100;
   Program.Landmark4 := FALSE;
   Program.Lifter4 := FALSE;
   Program.SpareBit1H4 := FALSE;
   Program.Airblower4 := TRUE;
   Program.NextStep4 := TRUE;
   Program.PressureP4 := TRUE;
   Program.SpareByte2H4 := 16#00;
   Program.Revolution4 := 3;
   Program.RopeUnit4_1 := 16#02;
   Program.RopeUnit4_2 := 16#02;
   Program.FilmForce4 := 30;
   Program.FilmPrestretch4 := 200;
   Program.Spare3H4 := 0;
   Program.Spare64 := 0;
   Program.Spare65 := 0;
   Program.Spare66 := 0;
   Program.Spare67 := 0;
   Program.Spare68 := 0;
   Program.Overlap4_5 := 0;
   Program.Height5 := 50;
   Program.Landmark5 := FALSE;
   Program.Lifter5 := FALSE;
   Program.SpareBit1H5 := FALSE;
   Program.Airblower5 := TRUE;
   Program.NextStep5 := FALSE;
   Program.PressureP5 := FALSE;
   Program.SpareByte2H5 := 16#00;
   Program.Revolution5 := 1;
   Program.RopeUnit5_1 := 16#01;
   Program.RopeUnit5_2 := 16#01;
   Program.FilmForce5 := 30;
   Program.FilmPrestretch5 := 200;
   Program.Spare3H5 := 0;
   Program.Spare69 := 0;
   Program.Spare70 := 0;
   Program.Spare71 := 0;
   Program.Spare72 := 0;
   Program.Spare73 := 0;
   Program.Overlap5_6 := 100;
   Program.Height6 := 50;
   Program.Landmark6 := FALSE;
   Program.Lifter6 := FALSE;
   Program.SpareBit1H6 := FALSE;
   Program.Airblower6 := TRUE;
   Program.NextStep6 := FALSE;
   Program.PressureP6 := FALSE;
   Program.SpareByte2H6 := 16#00;
   Program.Revolution6 := 2;
   Program.RopeUnit6_1 := 16#02;
   Program.RopeUnit6_2 := 16#01;
   Program.FilmForce6 := 20;
   Program.FilmPrestretch6 := 200;
   Program.Spare3H6 := 0;
   Program.Spare74 := 0;
   Program.Spare75 := 0;
   Program.Spare76 := 0;
   Program.Spare77 := 0;
   Program.Spare78 := 0;
   Program.Overlap6_7 := 0;
   Program.Height7 := 0;
   Program.Landmark7 := FALSE;
   Program.Lifter7 := FALSE;
   Program.SpareBit1H7 := FALSE;
   Program.Airblower7 := FALSE;
   Program.NextStep7 := TRUE;
   Program.PressureP7 := FALSE;
   Program.SpareByte2H7 := 16#00;
   Program.Revolution7 := 1;
   Program.RopeUnit7_1 := 16#01;
   Program.RopeUnit7_2 := 16#01;
   Program.FilmForce7 := 0;
   Program.FilmPrestretch7 := 100;
   Program.Spare3H7 := 0;
   Program.Spare79 := 0;
   Program.Spare80 := 0;
   Program.Spare81 := 0;
   Program.Spare82 := 0;
   Program.Spare83 := 0;
   Program.Overlap7_8 := 0;
   Program.Height8 := 0;
   Program.Landmark8 := FALSE;
   Program.Lifter8 := FALSE;
   Program.SpareBit1H8 := FALSE;
   Program.Airblower8 := FALSE;
   Program.NextStep8 := TRUE;
   Program.PressureP8 := FALSE;
   Program.SpareByte2H8 := 16#00;
   Program.Revolution8 := 1;
   Program.RopeUnit8_1 := 16#01;
   Program.RopeUnit8_2 := 16#01;
   Program.FilmForce8 := 0;
   Program.FilmPrestretch8 := 100;
   Program.Spare3H8 := 0;
   Program.Spare84 := 0;
   Program.Spare85 := 0;
   Program.Spare86 := 0;
   Program.Spare87 := 0;
   Program.Spare88 := 0;
   Program.Overlap8_9 := 0;
   Program.Height9 := 0;
   Program.Landmark9 := FALSE;
   Program.Lifter9 := FALSE;
   Program.SpareBit1H9 := FALSE;
   Program.Airblower9 := FALSE;
   Program.NextStep9 := TRUE;
   Program.PressureP9 := FALSE;
   Program.SpareByte2H9 := 16#00;
   Program.Revolution9 := 1;
   Program.RopeUnit9_1 := 16#01;
   Program.RopeUnit9_2 := 16#01;
   Program.FilmForce9 := 0;
   Program.FilmPrestretch9 := 100;
   Program.Spare3H9 := 0;
   Program.Spare89 := 0;
   Program.Spare90 := 0;
   Program.Spare91 := 0;
   Program.Spare92 := 0;
   Program.Spare93 := 0;
   Program.Overlap9_10 := 0;
   Program.Height10 := 0;
   Program.Landmark10 := FALSE;
   Program.Lifter10 := FALSE;
   Program.SpareBit1H10 := FALSE;
   Program.Airblower10 := FALSE;
   Program.NextStep10 := FALSE;
   Program.PressureP10 := FALSE;
   Program.SpareByte2H10 := 16#00;
   Program.Revolution10 := 1;
   Program.RopeUnit10_1 := 16#01;
   Program.RopeUnit10_2 := 16#01;
   Program.FilmForce10 := 0;
   Program.FilmPrestretch10 := 100;
   Program.Spare3H10 := 0;
   Program.Spare94 := 0;
   Program.Spare95 := 0;
   Program.Spare96 := 0;
   Program.Spare97 := 0;
   Program.Spare98 := 0;
   Program.Overlap10_11 := 0;
   Program.Height11 := 0;
   Program.Landmark11 := FALSE;
   Program.Lifter11 := FALSE;
   Program.SpareBit1H11 := FALSE;
   Program.Airblower11 := FALSE;
   Program.NextStep11 := TRUE;
   Program.PressureP11 := FALSE;
   Program.SpareByte2H11 := 16#00;
   Program.Revolution11 := 1;
   Program.RopeUnit11_1 := 16#01;
   Program.RopeUnit11_2 := 16#01;
   Program.FilmForce11 := 0;
   Program.FilmPrestretch11 := 100;
   Program.Spare3H11 := 0;
   Program.Spare99 := 0;
   Program.Spare100 := 0;
   Program.Spare101 := 0;
   Program.Spare102 := 0;
   Program.Spare103 := 0;
   Program.Overlap11_12 := 0;
   Program.Height12 := 0;
   Program.Landmark12 := FALSE;
   Program.Lifter12 := FALSE;
   Program.SpareBit1H12 := FALSE;
   Program.Airblower12 := FALSE;
   Program.NextStep12 := FALSE;
   Program.PressureP12 := FALSE;
   Program.SpareByte2H12 := 16#00;
   Program.Revolution12 := 1;
   Program.RopeUnit12_1 := 16#01;
   Program.RopeUnit12_2 := 16#01;
   Program.FilmForce12 := 0;
   Program.FilmPrestretch12 := 100;
   Program.Spare3H12 := 0;
   Program.Spare104 := 0;
   Program.Spare105 := 0;
   Program.Spare106 := 0;
   Program.Spare107 := 0;
   Program.Spare108 := 0;
END_DATA_BLOCK

DATA_BLOCK "DB251_ProgramDisplay"   // DB251
{ S7_Optimized_Access := 'FALSE' }
VERSION : 0.0
// stored: AutoNumber false, IsOnlyStoredInLoadMemory false, IsWriteProtectedInAS false
   VAR RETAIN
      Display { S7_SetPoint := 'True'} : "DatiProgramma";
   END_VAR
BEGIN
   Display.Wrapping := TRUE;
   Display.TopLenght := 500;
   Display.TopRelease := 0;
   Display.TopDown := 0;
   Display.Top := 4;
   Display.PressurePTime := 0;
   Display.LifterTime := 0;
   Display.RevOverContrast := 1;
   Display.RopeEndCycle := 16#02;
   Display.Spare4 := 16#01;
   Display.RopeTime := 1500;
   Display.RevOverClamp := 1;
   Display.FilmForceFinalRev := 10;
   Display.FilmPrestretchFinalRev := 100;
   Display.ArmSpeed := 100;
   Display.CarriageDown4Top := 500;
   Display.TopDownTime := 1500;
   Display.LapsUnderTop := 0;
   Display.Spare6 := 0;
   Display.Spare7 := 0;
   Display.Spare8 := 0;
   Display.Spare9 := 0;
   Display.Spare10 := 0;
   Display.Spare11 := 0;
   Display.Spare12 := 0;
   Display.Overlap0_1 := 0;
   Display.Height1 := 130;
   Display.Landmark1 := FALSE;
   Display.Lifter1 := FALSE;
   Display.SpareBit1H1 := FALSE;
   Display.Airblower1 := TRUE;
   Display.NextStep1 := TRUE;
   Display.PressureP1 := TRUE;
   Display.SpareByte2H1 := 16#00;
   Display.Revolution1 := 1;
   Display.RopeUnit1_1 := 16#01;
   Display.RopeUnit1_2 := 16#01;
   Display.FilmForce1 := 5;
   Display.FilmPrestretch1 := 200;
   Display.Spare3H1 := 0;
   Display.Spare49 := 0;
   Display.Spare50 := 0;
   Display.Spare51 := 0;
   Display.Spare52 := 0;
   Display.Spare53 := 0;
   Display.Overlap1_2 := 0;
   Display.Height2 := 50;
   Display.Landmark2 := FALSE;
   Display.Lifter2 := FALSE;
   Display.SpareBit1H2 := FALSE;
   Display.Airblower2 := TRUE;
   Display.NextStep2 := TRUE;
   Display.PressureP2 := TRUE;
   Display.SpareByte2H2 := 16#00;
   Display.Revolution2 := 1;
   Display.RopeUnit2_1 := 16#01;
   Display.RopeUnit2_2 := 16#01;
   Display.FilmForce2 := 20;
   Display.FilmPrestretch2 := 200;
   Display.Spare3H2 := 0;
   Display.Spare54 := 0;
   Display.Spare55 := 0;
   Display.Spare56 := 0;
   Display.Spare57 := 0;
   Display.Spare58 := 0;
   Display.Overlap2_3 := 100;
   Display.Height3 := -50;
   Display.Landmark3 := TRUE;
   Display.Lifter3 := FALSE;
   Display.SpareBit1H3 := FALSE;
   Display.Airblower3 := TRUE;
   Display.NextStep3 := TRUE;
   Display.PressureP3 := TRUE;
   Display.SpareByte2H3 := 16#00;
   Display.Revolution3 := 2;
   Display.RopeUnit3_1 := 16#01;
   Display.RopeUnit3_2 := 16#01;
   Display.FilmForce3 := 30;
   Display.FilmPrestretch3 := 200;
   Display.Spare3H3 := 0;
   Display.Spare59 := 0;
   Display.Spare60 := 0;
   Display.Spare61 := 380;
   Display.Spare62 := 2800;
   Display.Spare63 := 0;
   Display.Overlap3_4 := 100;
   Display.Height4 := 100;
   Display.Landmark4 := FALSE;
   Display.Lifter4 := FALSE;
   Display.SpareBit1H4 := FALSE;
   Display.Airblower4 := TRUE;
   Display.NextStep4 := TRUE;
   Display.PressureP4 := TRUE;
   Display.SpareByte2H4 := 16#00;
   Display.Revolution4 := 3;
   Display.RopeUnit4_1 := 16#02;
   Display.RopeUnit4_2 := 16#02;
   Display.FilmForce4 := 30;
   Display.FilmPrestretch4 := 200;
   Display.Spare3H4 := 0;
   Display.Spare64 := 0;
   Display.Spare65 := 0;
   Display.Spare66 := 0;
   Display.Spare67 := 0;
   Display.Spare68 := 0;
   Display.Overlap4_5 := 0;
   Display.Height5 := 50;
   Display.Landmark5 := FALSE;
   Display.Lifter5 := FALSE;
   Display.SpareBit1H5 := FALSE;
   Display.Airblower5 := TRUE;
   Display.NextStep5 := FALSE;
   Display.PressureP5 := FALSE;
   Display.SpareByte2H5 := 16#00;
   Display.Revolution5 := 1;
   Display.RopeUnit5_1 := 16#01;
   Display.RopeUnit5_2 := 16#01;
   Display.FilmForce5 := 30;
   Display.FilmPrestretch5 := 200;
   Display.Spare3H5 := 0;
   Display.Spare69 := 0;
   Display.Spare70 := 0;
   Display.Spare71 := 0;
   Display.Spare72 := 0;
   Display.Spare73 := 0;
   Display.Overlap5_6 := 100;
   Display.Height6 := 50;
   Display.Landmark6 := FALSE;
   Display.Lifter6 := FALSE;
   Display.SpareBit1H6 := FALSE;
   Display.Airblower6 := TRUE;
   Display.NextStep6 := FALSE;
   Display.PressureP6 := FALSE;
   Display.SpareByte2H6 := 16#00;
   Display.Revolution6 := 2;
   Display.RopeUnit6_1 := 16#02;
   Display.RopeUnit6_2 := 16#01;
   Display.FilmForce6 := 20;
   Display.FilmPrestretch6 := 200;
   Display.Spare3H6 := 0;
   Display.Spare74 := 0;
   Display.Spare75 := 0;
   Display.Spare76 := 0;
   Display.Spare77 := 0;
   Display.Spare78 := 0;
   Display.Overlap6_7 := 0;
   Display.Height7 := 0;
   Display.Landmark7 := FALSE;
   Display.Lifter7 := FALSE;
   Display.SpareBit1H7 := FALSE;
   Display.Airblower7 := FALSE;
   Display.NextStep7 := TRUE;
   Display.PressureP7 := FALSE;
   Display.SpareByte2H7 := 16#00;
   Display.Revolution7 := 1;
   Display.RopeUnit7_1 := 16#01;
   Display.RopeUnit7_2 := 16#01;
   Display.FilmForce7 := 0;
   Display.FilmPrestretch7 := 100;
   Display.Spare3H7 := 0;
   Display.Spare79 := 0;
   Display.Spare80 := 0;
   Display.Spare81 := 0;
   Display.Spare82 := 0;
   Display.Spare83 := 0;
   Display.Overlap7_8 := 0;
   Display.Height8 := 0;
   Display.Landmark8 := FALSE;
   Display.Lifter8 := FALSE;
   Display.SpareBit1H8 := FALSE;
   Display.Airblower8 := FALSE;
   Display.NextStep8 := TRUE;
   Display.PressureP8 := FALSE;
   Display.SpareByte2H8 := 16#00;
   Display.Revolution8 := 1;
   Display.RopeUnit8_1 := 16#01;
   Display.RopeUnit8_2 := 16#01;
   Display.FilmForce8 := 0;
   Display.FilmPrestretch8 := 100;
   Display.Spare3H8 := 0;
   Display.Spare84 := 0;
   Display.Spare85 := 0;
   Display.Spare86 := 0;
   Display.Spare87 := 0;
   Display.Spare88 := 0;
   Display.Overlap8_9 := 0;
   Display.Height9 := 0;
   Display.Landmark9 := FALSE;
   Display.Lifter9 := FALSE;
   Display.SpareBit1H9 := FALSE;
   Display.Airblower9 := FALSE;
   Display.NextStep9 := TRUE;
   Display.PressureP9 := FALSE;
   Display.SpareByte2H9 := 16#00;
   Display.Revolution9 := 1;
   Display.RopeUnit9_1 := 16#01;
   Display.RopeUnit9_2 := 16#01;
   Display.FilmForce9 := 0;
   Display.FilmPrestretch9 := 100;
   Display.Spare3H9 := 0;
   Display.Spare89 := 0;
   Display.Spare90 := 0;
   Display.Spare91 := 0;
   Display.Spare92 := 0;
   Display.Spare93 := 0;
   Display.Overlap9_10 := 0;
   Display.Height10 := 0;
   Display.Landmark10 := FALSE;
   Display.Lifter10 := FALSE;
   Display.SpareBit1H10 := FALSE;
   Display.Airblower10 := FALSE;
   Display.NextStep10 := FALSE;
   Display.PressureP10 := FALSE;
   Display.SpareByte2H10 := 16#00;
   Display.Revolution10 := 1;
   Display.RopeUnit10_1 := 16#01;
   Display.RopeUnit10_2 := 16#01;
   Display.FilmForce10 := 0;
   Display.FilmPrestretch10 := 100;
   Display.Spare3H10 := 0;
   Display.Spare94 := 0;
   Display.Spare95 := 0;
   Display.Spare96 := 0;
   Display.Spare97 := 0;
   Display.Spare98 := 0;
   Display.Overlap10_11 := 0;
   Display.Height11 := 0;
   Display.Landmark11 := FALSE;
   Display.Lifter11 := FALSE;
   Display.SpareBit1H11 := FALSE;
   Display.Airblower11 := FALSE;
   Display.NextStep11 := TRUE;
   Display.PressureP11 := FALSE;
   Display.SpareByte2H11 := 16#00;
   Display.Revolution11 := 1;
   Display.RopeUnit11_1 := 16#01;
   Display.RopeUnit11_2 := 16#01;
   Display.FilmForce11 := 0;
   Display.FilmPrestretch11 := 100;
   Display.Spare3H11 := 0;
   Display.Spare99 := 0;
   Display.Spare100 := 0;
   Display.Spare101 := 0;
   Display.Spare102 := 0;
   Display.Spare103 := 0;
   Display.Overlap11_12 := 0;
   Display.Height12 := 0;
   Display.Landmark12 := FALSE;
   Display.Lifter12 := FALSE;
   Display.SpareBit1H12 := FALSE;
   Display.Airblower12 := FALSE;
   Display.NextStep12 := FALSE;
   Display.PressureP12 := FALSE;
   Display.SpareByte2H12 := 16#00;
   Display.Revolution12 := 1;
   Display.RopeUnit12_1 := 16#01;
   Display.RopeUnit12_2 := 16#01;
   Display.FilmForce12 := 0;
   Display.FilmPrestretch12 := 100;
   Display.Spare3H12 := 0;
   Display.Spare104 := 0;
   Display.Spare105 := 0;
   Display.Spare106 := 0;
   Display.Spare107 := 0;
   Display.Spare108 := 0;
END_DATA_BLOCK

DATA_BLOCK "DB320_PID"   // DB320
TITLE = PID
{ S7_Optimized_Access := 'FALSE' }
VERSION : 0.1
// stored: AutoNumber false, IsOnlyStoredInLoadMemory false, IsWriteProtectedInAS false
   VAR RETAIN
      PID { S7_SetPoint := 'True'} : "PID";
   END_VAR
BEGIN
   PID.proporzionale := 0;
   PID.integrativo := 0;
   PID.segnale := 0;
   PID.maxSegnale := 1000;
   PID.minSegnale := 0;
   PID.setPointShow := 265;
   PID.tiro := 0;
   PID.vParP := 70;
   PID.vParI := 70;
   PID.svuota := TRUE;
   PID.attiva := TRUE;
   PID.setTiro := FALSE;
   PID."timer" := T#0MS;
END_DATA_BLOCK

DATA_BLOCK "DB322_APP"   // DB322
TITLE = PID
{ S7_Optimized_Access := 'FALSE' }
VERSION : 0.1
// stored: AutoNumber false, IsOnlyStoredInLoadMemory false, IsWriteProtectedInAS false
   VAR RETAIN
      IN0 : Int := 0;
      IN1 : Int := 0;
      IN2 : Int := 0;
      IN3 : Int := 0;
      IN4 : Int := 0;
      IN5 : Int := 0;
      IN6 : Int := 0;
      IN7 : Int := 0;
      IN8 : Int := 0;
      IN9 : Int := 0;
      IN10 : DInt := 224;
      IN11 : DInt := 240;
      IN12 : DInt := 0;   // TIRO EQUIVALENTE SU CELLA (kg)
      APP { S7_SetPoint := 'True'} : "APP";
   END_VAR
BEGIN
   APP.PID_ComponenteProporzionale := 0;
   APP.PID_ComponenteIntegrale := 0;
   APP.PID_ComponenteDerivativa := 0;
   APP.Tiro := 0;
   APP.Tiro1 := 0;
   APP.Tiro2 := 0;
   APP.TiroPrecedente := 0;
   APP.TiroAppoggio := 0;
   APP.ErroreAttuale := 0;
   APP.ErrorePrecedente := 0;
   APP.PID_Kp := 70;
   APP.PID_Ki := 60;
   APP.PID_Kd := 0;
   APP.SetpointTiro := 56;
   APP.SetpointTiroRampa := 750;
   APP.TransitorioInizialeFase1 := 0;
   APP.TransitorioFase3 := 1;
   APP.TransitorioFase4 := 1;
   APP.VelocitaRotazione := 5;
   APP.VelocitaRotazioneFase2 := 100;
   APP.VelocitaRotazioneAppoggio1 := 100;
   APP.VelocitaRotazioneAppoggio2 := 100;
   APP.Fase1OneShoot := 0;
   APP.Fase2OneShoot := 0;
   APP.Fase3OneShoot := 0;
   APP.Fase4OneShoot := 0;
   APP.ArrestoRepentinoOneShoot := 0;
   APP.TiroFase1 := 0;
   APP.TempIntero := 90;
   APP.Fase := 0;
   APP.BallerinoPrecedente[0..2] := 56;
   APP.LimiteComponenteIntegrale := 20000;
   APP.TiroRichiesto := 10;
   APP.TimerArrestoRepentino := 2;
   APP.TiroMinimoArrestoRepentino := 10;
   APP.VariazioneTiro := 0;
   APP.TimerFase2 := 0;
   APP.TempoRotturaFilm := 166;
   APP.TimerFase4 := 0;
   APP.TiroMinimoFase4 := 6;
   APP.PID_Uscita := 0;
   APP.PrestiroRichiesto := 300;
   APP.PrestiroAppoggio := 0.5;
END_DATA_BLOCK

DATA_BLOCK "DB50_Config"   // DB50
{ S7_Optimized_Access := 'FALSE' }
VERSION : 0.1
// stored: AutoNumber false, IsOnlyStoredInLoadMemory false, IsWriteProtectedInAS false
   VAR RETAIN
      Sel1_Clamp : Int := 3;
      Sel2_BarrierIn : Int := 2;
      Sel3_Pressure : Int := 1;
      Sel4_Doors : Int := 0;
      Sel5_Carriage : Int := 1;
      Sel6_Selfcenter : Int := 2;
      Sel7_Top : Int := 1;
      Sel8_Rope : Int := 3;
      Sel9_BarrierOut : Int := 2;
      Sel10_Conv : Int := 16;
      Sel_Door : Bool := TRUE;
      Sel_EsaurFilm : Bool := FALSE;
      Sel_spare_bool_1 : Bool := FALSE;
      Sel_spare_bool_2 : Bool := FALSE;
      Sel_spare_bool_3 : Bool := FALSE;
      Sel_spare_bool_4 : Bool := FALSE;
      Sel_spare_bool_5 : Bool := FALSE;
      Sel_spare10 : Byte := 16#00;
      Sel_spare11 : Int := 0;
      Sel_spare12 : Int := 0;
      Sel_spare13 : Int := 0;
      Sel_spare14 : Int := 0;
      Sel_spare15 : Int := 0;
      Sel_spare16 : Int := 0;
      Sel_spare17 : Int := 0;
      Sel_spare18 : Int := 0;
      Sel_spare19 : Int := 0;
      Sel_spare20 : Int := 0;
      Sel_spare21 : Int := 0;
      Sel_spare22 : Int := 0;
      Sel_spare23 : Int := 0;
      Sel_spare24 : Int := 0;
      TimerPageFw : Bool := FALSE;
      TimerPageBkw : Bool := FALSE;
   END_VAR
BEGIN
END_DATA_BLOCK

DATA_BLOCK "DB80_Label"   // DB80
{ S7_Optimized_Access := 'FALSE' }
VERSION : 0.1
// stored: AutoNumber false, IsOnlyStoredInLoadMemory false, IsWriteProtectedInAS false
   VAR RETAIN
      Step0 : Bool := FALSE;   // Table rotation to first label position
      Step1 : Bool := FALSE;   // First label apply
      Step2 : Bool := FALSE;   // Table rotation to second label position
      Step3 : Bool := FALSE;   // Second label apply
      Step4 : Bool := FALSE;   // Table rotation to third label position
      Step5 : Bool := FALSE;   // Third label apply
      Step6 : Bool := FALSE;   // Table rotation to fourth label position
      Step7 : Bool := FALSE;   // Fourt label apply
      Step8 : Bool := FALSE;   // Table rotation to end cycle position
      spare_Step9 : Bool := FALSE;
      spare_Step10 : Bool := FALSE;
      spare_Step11 : Bool := FALSE;
      spare_Step12 : Bool := FALSE;
      spare_Step13 : Bool := FALSE;
      spare_Step14 : Bool := FALSE;
      spare_Step15 : Bool := FALSE;
      Phase1_On : Bool := TRUE;
      Phase2_On : Bool := FALSE;
      Phase3_On : Bool := TRUE;
      Phase4_On : Bool := FALSE;
      Enable : Bool := TRUE;
      rotation : Bool := FALSE;   // Table rotation for label command
      label_ok1 : Bool := FALSE;   // Label cycle ended
      S1 : Bool := FALSE;   // Label request signal
      spare_signal2 : Bool := FALSE;
      spare_signal3 : Bool := FALSE;
      spare_signal4 : Bool := FALSE;
      spare_signal5 : Bool := FALSE;
      spare_signal6 : Bool := FALSE;
      spare_signal7 : Bool := FALSE;
      spare_signal8 : Bool := FALSE;
      E1 : Bool := TRUE;   // Label arm in home position for pallet transit
      E2 : Bool := FALSE;   // Label applied signal
      E3 : Bool := FALSE;   // Label fault signal
      spare_input4 : Bool := FALSE;
      spare_input5 : Bool := FALSE;
      spare_input6 : Bool := FALSE;
      spare_input7 : Bool := FALSE;
      spare_input8 : Bool := FALSE;
      spare_byte5 : Byte := 16#00;
      Phase1 : Int := 900;
      Phase2 : Int := 1800;
      Phase3 : Int := 2700;
      Phase4 : Int := 3600;
      NextPhase : Int := 2700;
   END_VAR
BEGIN
END_DATA_BLOCK

DATA_BLOCK "DB88_Top"   // DB88
{ S7_Optimized_Access := 'FALSE' }
AUTHOR : Robopac
VERSION : 0.0
// stored: AutoNumber false, IsOnlyStoredInLoadMemory false, IsWriteProtectedInAS false
   VAR RETAIN
      VW800 : Int := 0;
      VW802 : Int := 0;
      V804_0 : Bool := FALSE;   // Top carriage in cut position
      V804_1 : Bool := FALSE;   // Top carriage in forward position
      V804_2 : Bool := FALSE;
      V804_3 : Bool := FALSE;   // Memory to stop top carriage forward in manual mode
      V804_4 : Bool := FALSE;   // Memory for top cut done
      V804_5 : Bool := FALSE;
      V804_6 : Bool := FALSE;
      V804_7 : Bool := FALSE;
      VB805 : Byte := 16#00;
      VW806 : Int := 0;   // Top positioning counter
   END_VAR
BEGIN
END_DATA_BLOCK

DATA_BLOCK "DeviceStates"   // DB12
{ S7_Optimized_Access := 'FALSE' }
VERSION : 0.1
// stored: AutoNumber true, IsOnlyStoredInLoadMemory false, IsWriteProtectedInAS false
   VAR
      LADDR : HW_IOSYSTEM := 16#010F;
      MODE : UInt := 4;
      returnValue : Int := 0;
      STATE : Array[0..1023] of Bool;
   END_VAR
BEGIN
   STATE[0..3] := TRUE;
   STATE[4..1023] := FALSE;
END_DATA_BLOCK

DATA_BLOCK "Inverter_Data"   // DB210
{ S7_Optimized_Access := 'FALSE' }
VERSION : 0.1
// stored: AutoNumber false, IsOnlyStoredInLoadMemory false, IsWriteProtectedInAS false
   VAR
      U201 { S7_SetPoint := 'True'} : "InverterData";
      U221 { S7_SetPoint := 'True'} : "InverterData";
      U241 { S7_SetPoint := 'True'} : "InverterData";
      U261 { S7_SetPoint := 'True'} : "InverterData";
      U321 { S7_SetPoint := 'True'} : "InverterData";
   END_VAR
BEGIN
   U201.control_word := 16#047A;
   U201.setpoint := 0.0;
   U201.ref_quantity.speed_p2000 := 3000.0;
   U201.ref_quantity.current_p2002 := 5.0;
   U201.ref_quantity.torque_p2003 := 7.61;
   U201.status_word := 16#EB40;
   U201.actual_speed := 0.0;
   U201.actual_current := 0.0;
   U201.actual_torque := 0.0;
   U201.actual_alarm := 16#0000;
   U201.actual_fault := 16#0000;
   U201.RETVAL_RD := 16#0000;
   U201.RETVAL_WR := 16#0000;
   U221.control_word := 16#047E;
   U221.setpoint := 0.0;
   U221.ref_quantity.speed_p2000 := 3000.0;
   U221.ref_quantity.current_p2002 := 1.86;
   U221.ref_quantity.torque_p2003 := 3.59;
   U221.status_word := 16#EB31;
   U221.actual_speed := 0.0;
   U221.actual_current := 0.001702881;
   U221.actual_torque := 0.0;
   U221.actual_alarm := 16#0000;
   U221.actual_fault := 16#0000;
   U221.RETVAL_RD := 16#0000;
   U221.RETVAL_WR := 16#0000;
   U241.control_word := 16#047E;
   U241.setpoint := 0.0;
   U241.ref_quantity.speed_p2000 := 3000.0;
   U241.ref_quantity.current_p2002 := 1.86;
   U241.ref_quantity.torque_p2003 := 3.59;
   U241.status_word := 16#EB31;
   U241.actual_speed := 0.0;
   U241.actual_current := 0.002043457;
   U241.actual_torque := 0.0;
   U241.actual_alarm := 16#0000;
   U241.actual_fault := 16#0000;
   U241.RETVAL_RD := 16#0000;
   U241.RETVAL_WR := 16#0000;
   U261.control_word := 16#047E;
   U261.setpoint := 0.0;
   U261.ref_quantity.speed_p2000 := 3000.0;
   U261.ref_quantity.current_p2002 := 1.86;
   U261.ref_quantity.torque_p2003 := 3.59;
   U261.status_word := 16#EB31;
   U261.actual_speed := 0.0;
   U261.actual_current := 0.0;
   U261.actual_torque := 0.0;
   U261.actual_alarm := 16#0000;
   U261.actual_fault := 16#0000;
   U261.RETVAL_RD := 16#0000;
   U261.RETVAL_WR := 16#0000;
   U321.control_word := 16#047E;
   U321.setpoint := 0.0;
   U321.ref_quantity.speed_p2000 := 3000.0;
   U321.ref_quantity.current_p2002 := 6.9;
   U321.ref_quantity.torque_p2003 := 29.5;
   U321.status_word := 16#EB31;
   U321.actual_speed := 0.0;
   U321.actual_current := 0.0;
   U321.actual_torque := 0.0;
   U321.actual_alarm := 16#0000;
   U321.actual_fault := 16#0000;
   U321.RETVAL_RD := 16#0000;
   U321.RETVAL_WR := 16#0000;
END_DATA_BLOCK

DATA_BLOCK "Timer"   // DB2
{ S7_Optimized_Access := 'TRUE' }
VERSION : 0.0
// stored: AutoNumber false, IsOnlyStoredInLoadMemory false, IsRetainMemResEnabled false, IsWriteProtectedInAS false, MemoryReserve 100
   VAR
      T0 { S7_SetPoint := 'True'} : IEC_TIMER;   // Delay on pallet positioning
      T1 { S7_SetPoint := 'True'} : IEC_TIMER;   // Timer for acoustic siren
      T2 { S7_SetPoint := 'True'} : IEC_TIMER;   // Timer for restart after emergency
      T3 { S7_SetPoint := 'True'} : IEC_TIMER;   // Timer to reset emergency
      T4 { S7_SetPoint := 'True'} : IEC_TIMER;   // Timer to reset the cycles
      T5 { S7_SetPoint := 'True'} : IEC_TIMER;   // Delay for backward on table rotation inverter
      T6 { S7_SetPoint := 'True'} : IEC_TIMER;   // Delay for forward on table rotation inverter
      T7 { S7_SetPoint := 'True'} : IEC_TIMER;   // Timeout for table phase
      T8 { S7_SetPoint := 'True'} : IEC_TIMER;   // Table rotation speed timer
      T9 { S7_SetPoint := 'True'} : IEC_TIMER;   // Timer SA type for spool carriage motor
      T10 { S7_SetPoint := 'True'} : IEC_TIMER;   // Timer SA type for table rotation motor
      T11 { S7_SetPoint := 'True'} : IEC_TIMER;   // Timer SA type for spool carriage downward
      T12 { S7_SetPoint := 'True'} : IEC_TIMER;   // Timer SA type for spool carriage upward
      T13 { S7_SetPoint := 'True'} : IEC_TIMER;   // Timer SA type for top carriage motor
      T14 { S7_SetPoint := 'True'} : IEC_TIMER;   // Delay for forward on spool carriage and machine conveyor inverter
      T15 { S7_SetPoint := 'True'} : IEC_TIMER;   // Timer for lifter upward
      T16 { S7_SetPoint := 'True'} : IEC_TIMER;   // Timeout for pallet lifter upward/downward
      T17 { S7_SetPoint := 'True'} : IEC_TIMER;   // Time for pressure plate downward
      T18 { S7_SetPoint := 'True'} : IEC_TIMER;   // Timeout for pressure plate upward/downward
      T19 { S7_SetPoint := 'True'} : IEC_TIMER;   // Delay for backward on spool carriage and machine conveyor inverter
      T20 { S7_SetPoint := 'True'} : IEC_TIMER;   // Delay for table rotation deceleration
      T21 { S7_SetPoint := 'True'} : IEC_TIMER;   // Film broken delay for spool carriage
      T22 { S7_SetPoint := 'True'} : IEC_TIMER;   // Delay for pressure plate positioning on pallet
      T23 { S7_SetPoint := 'True'} : IEC_TIMER;   // Timer SA type for conveyor motor
      T24 { S7_SetPoint := 'True'} : IEC_TIMER;   // Delay on pallet positioning left
      T25 { S7_SetPoint := 'True'} : IEC_TIMER;   // Delay on machine conveyor stop
      T26 { S7_SetPoint := 'True'} : IEC_TIMER;   // Delay to load/unload pallet simultaneously
      T27 { S7_SetPoint := 'True'} : IEC_TIMER;   // Delay to have outfeed control free
      T28 { S7_SetPoint := 'True'} : IEC_TIMER;   // Timer for end of transfer signal
      T29 { S7_SetPoint := 'True'} : IEC_TIMER;   // Timer to check spool carriage encoder
      T30 { S7_SetPoint := 'True'} : IEC_TIMER;   // Timer to check spool carriage encoder
      T31 { S7_SetPoint := 'True'} : IEC_TIMER;   // Time to record spool carriage movement speed
      T32 { S7_SetPoint := 'True'} : IEC_TIMER;   // Timeout for single or lower(double) rope unit open/close
      T33 { S7_SetPoint := 'True'} : IEC_TIMER;   // Timer for outfeed rotating table control engaged
      T34 { S7_SetPoint := 'True'} : IEC_TIMER;   // Timer for prestretch restart
      T35 { S7_SetPoint := 'True'} : IEC_TIMER;   // Delay to open single or lower(double) rope unit
      T36 { S7_SetPoint := 'True'} : IEC_TIMER;   // Timeout for welder unit upward/downward
      T37 { S7_SetPoint := 'True'} : IEC_TIMER;   // Timeout for welder contrast downward
      T38 { S7_SetPoint := 'True'} : IEC_TIMER;   // Timeout for welder contrast upward
      T39 { S7_SetPoint := 'True'} : IEC_TIMER;   // Timeout for clamp upward/downward
      T40 { S7_SetPoint := 'True'} : IEC_TIMER;   // Timeout for clamp open/close
      T41 { S7_SetPoint := 'True'} : IEC_TIMER;   // Welding timer for welder
      T42 { S7_SetPoint := 'True'} : IEC_TIMER;   // Cutting timer
      T43 { S7_SetPoint := 'True'} : IEC_TIMER;   // Welder cooler timer
      T44 { S7_SetPoint := 'True'} : IEC_TIMER;   // Timer to check welder circuit 1 (current on)
      T45 { S7_SetPoint := 'True'} : IEC_TIMER;   // Timer to check welder circuit 2 (current off)
      T46 { S7_SetPoint := 'True'} : IEC_TIMER;   // Spring clamp up
      T47 { S7_SetPoint := 'True'} : IEC_TIMER;   // Welder contrast up
      T48 { S7_SetPoint := 'True'} : IEC_TIMER;   // Spring clamp open
      T49 { S7_SetPoint := 'True'} : IEC_TIMER;   // Welder and cut unit up
      T50 { S7_SetPoint := 'True'} : IEC_TIMER;   // Timer for encoder check
      T51 { S7_SetPoint := 'True'} : IEC_TIMER;   // Timer for display comunication control
      T52 { S7_SetPoint := 'True'} : IEC_TIMER;   // Timer to return to page 1 after 3 minutes
      T53 { S7_SetPoint := 'True'} : IEC_TIMER;   // Delay for test cycle
      T54 { S7_SetPoint := 'True'} : IEC_TIMER;   // Timer to reset infeed safety barrier
      T55 { S7_SetPoint := 'True'} : IEC_TIMER;   // Timer to reset infeed safety barrier
      T56 { S7_SetPoint := 'True'} : IEC_TIMER;   // Timer to reset outfeed safety barrier
      T57 { S7_SetPoint := 'True'} : IEC_TIMER;   // Timer to reset outfeed safety barrier
      T58 { S7_SetPoint := 'True'} : IEC_TIMER;   // Delay for infeed safety barrier muting photocell
      T59 { S7_SetPoint := 'True'} : IEC_TIMER;   // Delay for outfeed safety barrier muting photocell
      T60 { S7_SetPoint := 'True'} : IEC_TIMER;   // Delay for spool carriage downward for film tail
      T61 { S7_SetPoint := 'True'} : IEC_TIMER;   // Delay to open clamp during wrapping cycle
      T62 { S7_SetPoint := 'True'} : IEC_TIMER;   // Timer for table rotation forward on twist
      T63 { S7_SetPoint := 'True'} : IEC_TIMER;   // Timer SA type for top carriage upward
      T64 { S7_SetPoint := 'True'} : IEC_TIMER;   // Timer SA type for top carriage downward
      T65 { S7_SetPoint := 'True'} : IEC_TIMER;   // Delay on safety for top carriage movement
      T66 { S7_SetPoint := 'True'} : IEC_TIMER;   // Timer to check top film presence
      T67 { S7_SetPoint := 'True'} : IEC_TIMER;   // Timer to check top film presence
      T68 { S7_SetPoint := 'True'} : IEC_TIMER;   // Timeout for top film cutter forward/backward
      T69 { S7_SetPoint := 'True'} : IEC_TIMER;   // Timeout for clamp to lift top film open/close
      T70 { S7_SetPoint := 'True'} : IEC_TIMER;   // Timeout for clamp to block top film open/close
      T71 { S7_SetPoint := 'True'} : IEC_TIMER;   // Timeout for top carriage forward/backward movement
      T72 { S7_SetPoint := 'True'} : IEC_TIMER;   // Timeout for top carriage forward/backward movement
      T73 { S7_SetPoint := 'True'} : IEC_TIMER;   // Timeout for top carriage upward/downward movement
      T74 { S7_SetPoint := 'True'} : IEC_TIMER;   // Timeout for top carriage upward/downward movement
      T75 { S7_SetPoint := 'True'} : IEC_TIMER;   // Delay for spool carriage downward during top cycle
      T76 { S7_SetPoint := 'True'} : IEC_TIMER;   // Claw clamp closed
      T77 { S7_SetPoint := 'True'} : IEC_TIMER;   // Timeout for welder and cut unit forward/backward
      T78 { S7_SetPoint := 'True'} : IEC_TIMER;   // Delay to open upper(double) rope unit
      T79 { S7_SetPoint := 'True'} : IEC_TIMER;   // Timer SA type for table rotation brake
      T80 { S7_SetPoint := 'True'} : IEC_TIMER;   // Timer for spool carriage movement speed
      T81 { S7_SetPoint := 'True'} : IEC_TIMER;   // Claw clamp closed
      T82 { S7_SetPoint := 'True'} : IEC_TIMER;   // Timeout for welder and cut unit forward/backward
      T83 { S7_SetPoint := 'True'} : IEC_TIMER;   // Delay between airblow and clamp
      T84 { S7_SetPoint := 'True'} : IEC_TIMER;   // Timer for table rotation speed
      T85 { S7_SetPoint := 'True'} : IEC_TIMER;   // Delay on infeed conveyor stop
      T86 { S7_SetPoint := 'True'} : IEC_TIMER;   // Delay for prestretch during acceleration
      T87 { S7_SetPoint := 'True'} : IEC_TIMER;   // Timer for slow conveyor manual movement
      T88 { S7_SetPoint := 'True'} : IEC_TIMER;
      T89 { S7_SetPoint := 'True'} : IEC_TIMER;   // Timer for wrong pallet positioning without outfeed control
      T90 { S7_SetPoint := 'True'} : IEC_TIMER;   // Timer for spool carriage upward for table cycle
      T91 { S7_SetPoint := 'True'} : IEC_TIMER;   // Delay to close clamp after cutter forward
      T92 { S7_SetPoint := 'True'} : IEC_TIMER;   // Delay for contrast downward
      T93 { S7_SetPoint := 'True'} : IEC_TIMER;
      T94 { S7_SetPoint := 'True'} : IEC_TIMER;
      T95 { S7_SetPoint := 'True'} : IEC_TIMER;
      T96 { S7_SetPoint := 'True'} : IEC_TIMER;   // Timeout for fire door pos.4-5 opening
      T97 { S7_SetPoint := 'True'} : IEC_TIMER;   // Delay conveyor manual movement
      T98 { S7_SetPoint := 'True'} : IEC_TIMER;   // Delay start cycle pos.1
      T99 { S7_SetPoint := 'True'} : IEC_TIMER;   // Time to load with forklift
      T100 { S7_SetPoint := 'True'} : IEC_TIMER;   // Timer for end of pallet transfer in infeed signal
      T101 { S7_SetPoint := 'True'} : IEC_TIMER;   // Timeout for conveyor pos 01
      T102 { S7_SetPoint := 'True'} : IEC_TIMER;   // Time to load with forklift
      T103 { S7_SetPoint := 'True'} : IEC_TIMER;   // Timeout for conveyor pos 02
      T104 { S7_SetPoint := 'True'} : IEC_TIMER;
      T105 { S7_SetPoint := 'True'} : IEC_TIMER;   // Timeout for conveyor pos 04
      T106 { S7_SetPoint := 'True'} : IEC_TIMER;   // Timeout for conveyor pos 03
      T107 { S7_SetPoint := 'True'} : IEC_TIMER;   // Time for pallet unload with forklift
      T108 { S7_SetPoint := 'True'} : IEC_TIMER;   // Delay Button Stop cycle support memory
      T109 { S7_SetPoint := 'True'} : IEC_TIMER;   // Time for pallet load with forklift from reverse
      T110 { S7_SetPoint := 'True'} : IEC_TIMER;   // Timer to reset machine and cycle
      T111 { S7_SetPoint := 'True'} : IEC_TIMER;   // Delay timer for lifter pos.2 low position
      T112 { S7_SetPoint := 'True'} : IEC_TIMER;   // Delay timer for lifter pos.2 up position
      T113 { S7_SetPoint := 'True'} : IEC_TIMER;   // Delay timer pallet positioned on lifter pos.2
      T114 { S7_SetPoint := 'True'} : IEC_TIMER;   // Timer SA for lifter in top position
      T115 { S7_SetPoint := 'True'} : IEC_TIMER;   // Timeout for conveyor pos.2
      T116 { S7_SetPoint := 'True'} : IEC_TIMER;   // Timeout for lifter pos.2 upstroke
      T117 { S7_SetPoint := 'True'} : IEC_TIMER;   // Timeout for lifter pos.2 downstroke
      T118 { S7_SetPoint := 'True'} : IEC_TIMER;   // Timer to filter lifter pos.2 in up position
      T119 { S7_SetPoint := 'True'} : IEC_TIMER;
      T120 { S7_SetPoint := 'True'} : IEC_TIMER;   // Timer to check conveyor encoder
      T121 { S7_SetPoint := 'True'} : IEC_TIMER;   // Timer to check conveyor encoder
      T122 { S7_SetPoint := 'True'} : IEC_TIMER;
      T123 { S7_SetPoint := 'True'} : IEC_TIMER;
      T124 { S7_SetPoint := 'True'} : IEC_TIMER;
      T125 { S7_SetPoint := 'True'} : IEC_TIMER;
      T126 { S7_SetPoint := 'True'} : IEC_TIMER;
      T127 { S7_SetPoint := 'True'} : IEC_TIMER;   // Delay to have outfeed rotating arm control free from reverse
      T128 { S7_SetPoint := 'True'} : IEC_TIMER;   // Timer for end of transfer signal from reverse
      T129 { S7_SetPoint := 'True'} : IEC_TIMER;
      T130 { S7_SetPoint := 'True'} : IEC_TIMER;
      T131 { S7_SetPoint := 'True'} : IEC_TIMER;
      T132 { S7_SetPoint := 'True'} : IEC_TIMER;   // Timeout for single or lower(double) rope unit open/close
      T133 { S7_SetPoint := 'True'} : IEC_TIMER;
      T134 { S7_SetPoint := 'True'} : IEC_TIMER;
      T135 { S7_SetPoint := 'True'} : IEC_TIMER;   // Delay to open single or lower(double) rope unit
      T136 { S7_SetPoint := 'True'} : IEC_TIMER;
      T137 { S7_SetPoint := 'True'} : IEC_TIMER;
      T138 { S7_SetPoint := 'True'} : IEC_TIMER;
      T139 { S7_SetPoint := 'True'} : IEC_TIMER;   // Delay for top carriage forward stop (Top)
      T140 { S7_SetPoint := 'True'} : IEC_TIMER;   // Delay for top carriage backward stop (Top)
      T141 { S7_SetPoint := 'True'} : IEC_TIMER;
      T142 { S7_SetPoint := 'True'} : IEC_TIMER;   // Delay for top carriage down to release top film (Top)
      T143 { S7_SetPoint := 'True'} : IEC_TIMER;   // Delay to release top film from clamp (Top)
      T144 { S7_SetPoint := 'True'} : IEC_TIMER;   // Timer 1 for top film broken (Top)
      T145 { S7_SetPoint := 'True'} : IEC_TIMER;   // Timer 2 for top film broken (Top)
      T146 { S7_SetPoint := 'True'} : IEC_TIMER;   // Delay to stop top carriage forward for top film broken (Top)
      T147 { S7_SetPoint := 'True'} : IEC_TIMER;   // Delay to stop top carriage against vibration (Top)
      T148 { S7_SetPoint := 'True'} : IEC_TIMER;   // Timeout for top cutter (Top)
      T149 { S7_SetPoint := 'True'} : IEC_TIMER;   // Timeout for clamp to pull top film (Top)
      T150 { S7_SetPoint := 'True'} : IEC_TIMER;   // Timeout for clamp to block top film (Top)
      T151 { S7_SetPoint := 'True'} : IEC_TIMER;   // Timer SA type for top brake (Top)
      T152 { S7_SetPoint := 'True'} : IEC_TIMER;   // Timer for top brake control (Top)
      T153 { S7_SetPoint := 'True'} : IEC_TIMER;
      T154 { S7_SetPoint := 'True'} : IEC_TIMER;
      T155 { S7_SetPoint := 'True'} : IEC_TIMER;   // Timeout for conveyor pos 03
      T156 { S7_SetPoint := 'True'} : IEC_TIMER;   // Timeout for conveyor pos 04
      T157 { S7_SetPoint := 'True'} : IEC_TIMER;   // Timeout for conveyor pos 05
      T158 { S7_SetPoint := 'True'} : IEC_TIMER;   // Timeout for conveyor pos 06
      T159 { S7_SetPoint := 'True'} : IEC_TIMER;   // Timeout for conveyor pos 07
      T160 { S7_SetPoint := 'True'} : IEC_TIMER;   // Timeout for conveyor pos 08
      T161 { S7_SetPoint := 'True'} : IEC_TIMER;
      T162 { S7_SetPoint := 'True'} : IEC_TIMER;
      T163 { S7_SetPoint := 'True'} : IEC_TIMER;   // Watchdog timer for network communication
      T164 { S7_SetPoint := 'True'} : IEC_TIMER;
      T165 { S7_SetPoint := 'True'} : IEC_TIMER;
      T166 { S7_SetPoint := 'True'} : IEC_TIMER;
      T167 { S7_SetPoint := 'True'} : IEC_TIMER;
      T168 { S7_SetPoint := 'True'} : IEC_TIMER;
      T169 { S7_SetPoint := 'True'} : IEC_TIMER;
      T170 { S7_SetPoint := 'True'} : IEC_TIMER;
      T171 { S7_SetPoint := 'True'} : IEC_TIMER;
      T172 { S7_SetPoint := 'True'} : IEC_TIMER;
      T173 { S7_SetPoint := 'True'} : IEC_TIMER;
      T174 { S7_SetPoint := 'True'} : IEC_TIMER;
      T175 { S7_SetPoint := 'True'} : IEC_TIMER;
      T176 { S7_SetPoint := 'True'} : IEC_TIMER;
      T177 { S7_SetPoint := 'True'} : IEC_TIMER;
      T178 { S7_SetPoint := 'True'} : IEC_TIMER;
      T179 { S7_SetPoint := 'True'} : IEC_TIMER;   // Delay for top pallet height reading photocell (fast cycle)
      T180 { S7_SetPoint := 'True'} : IEC_TIMER;
      T181 { S7_SetPoint := 'True'} : IEC_TIMER;
      T182 { S7_SetPoint := 'True'} : IEC_TIMER;
      T183 { S7_SetPoint := 'True'} : IEC_TIMER;
      T184 { S7_SetPoint := 'True'} : IEC_TIMER;
      T185 { S7_SetPoint := 'True'} : IEC_TIMER;
      T186 { S7_SetPoint := 'True'} : IEC_TIMER;
      T187 { S7_SetPoint := 'True'} : IEC_TIMER;
      T188 { S7_SetPoint := 'True'} : IEC_TIMER;
      T189 { S7_SetPoint := 'True'} : IEC_TIMER;
      T190 { S7_SetPoint := 'True'} : IEC_TIMER;
      T191 { S7_SetPoint := 'True'} : IEC_TIMER;
      T192 { S7_SetPoint := 'True'} : IEC_TIMER;
      T193 { S7_SetPoint := 'True'} : IEC_TIMER;
      T194 { S7_SetPoint := 'True'} : IEC_TIMER;
      T195 { S7_SetPoint := 'True'} : IEC_TIMER;
      T196 { S7_SetPoint := 'True'} : IEC_TIMER;
      T197 { S7_SetPoint := 'True'} : IEC_TIMER;
      T198 { S7_SetPoint := 'True'} : IEC_TIMER;
      T199 { S7_SetPoint := 'True'} : IEC_TIMER;
      T200 { S7_SetPoint := 'True'} : IEC_TIMER;   // T_InverterAlarm - Time to filter inverter alarms
      T201 { S7_SetPoint := 'True'} : IEC_TIMER;   // T_ProfinetDiag - Time to filter 'DeviceStates' diagnostic output (Profinet)
      T202 { S7_SetPoint := 'True'} : IEC_TIMER;   // Timer for U201 start command (after enable)
      T203 { S7_SetPoint := 'True'} : IEC_TIMER;   // Timer table backward
      T204 { S7_SetPoint := 'True'} : IEC_TIMER;   // Timer ciclo fiera
      T205 { S7_SetPoint := 'True'} : IEC_TIMER;   // TON per OFF1 U201
      T206 { S7_SetPoint := 'True'} : IEC_TIMER;   // TOF per OFF1 U201
      T207 { S7_SetPoint := 'True'} : IEC_TIMER;   // Timer coppia tavola
      T208 { S7_SetPoint := 'True'} : IEC_TIMER;   // T_ModbusErrors
      T209 { S7_SetPoint := 'True'} : IEC_TIMER;
      T210 { S7_SetPoint := 'True'} : IEC_TIMER;   // Time to filter contrast back sensor
      T211 { S7_SetPoint := 'True'} : IEC_TIMER;   // Timeout for welder contrast forward
      T212 { S7_SetPoint := 'True'} : IEC_TIMER;   // Timeout for welder contrast backward
      T213 { S7_SetPoint := 'True'} : IEC_TIMER;   // Timeout for (double) full rope unit open/close
      T214 { S7_SetPoint := 'True'} : IEC_TIMER;   // Delay to open single or lower(double) rope unit
      T215 { S7_SetPoint := 'True'} : IEC_TIMER;   // Time Contrast Backward
      T216 { S7_SetPoint := 'True'} : IEC_TIMER;   // Time Contrast Manual forward
   END_VAR
BEGIN
   T0.PT := T#0MS;
   T0.IN := FALSE;
   T1.PT := T#1S_200MS;
   T1.IN := FALSE;
   T2.PT := T#6S;
   T2.IN := TRUE;
   T3.PT := T#700MS;
   T3.IN := FALSE;
   T4.PT := T#2S;
   T4.IN := FALSE;
   T5.PT := T#800MS;
   T5.IN := FALSE;
   T6.PT := T#800MS;
   T6.IN := FALSE;
   T7.PT := T#50S;
   T7.IN := FALSE;
   T8.PT := T#1M_39S;
   T8.IN := FALSE;
   T9.PT := T#700MS;
   T9.IN := FALSE;
   T10.PT := T#2S;
   T10.IN := FALSE;
   T11.PT := T#500MS;
   T11.IN := FALSE;
   T12.PT := T#500MS;
   T12.IN := FALSE;
   T13.PT := T#0MS;
   T13.IN := FALSE;
   T14.PT := T#200MS;
   T14.IN := FALSE;
   T15.PT := T#0MS;
   T15.IN := FALSE;
   T16.PT := T#0MS;
   T16.IN := FALSE;
   T17.PT := T#0MS;
   T17.IN := FALSE;
   T18.PT := T#0MS;
   T18.IN := FALSE;
   T19.PT := T#200MS;
   T19.IN := FALSE;
   T20.PT := T#0MS;
   T20.IN := FALSE;
   T21.PT := T#2S;
   T21.IN := FALSE;
   T22.PT := T#0MS;
   T22.IN := FALSE;
   T23.PT := T#0MS;
   T23.IN := FALSE;
   T24.PT := T#0MS;
   T24.IN := FALSE;
   T25.PT := T#0MS;
   T25.IN := FALSE;
   T26.PT := T#0MS;
   T26.IN := FALSE;
   T27.PT := T#1S_500MS;
   T27.IN := TRUE;
   T28.PT := T#2S;
   T28.IN := TRUE;
   T29.PT := T#0MS;
   T29.IN := FALSE;
   T30.PT := T#3S;
   T30.IN := FALSE;
   T31.PT := T#0MS;
   T31.IN := FALSE;
   T32.PT := T#0MS;
   T32.IN := FALSE;
   T33.PT := T#0MS;
   T33.IN := FALSE;
   T34.PT := T#0MS;
   T34.IN := FALSE;
   T35.PT := T#0MS;
   T35.IN := FALSE;
   T36.PT := T#0MS;
   T36.IN := FALSE;
   T37.PT := T#0MS;
   T37.IN := FALSE;
   T38.PT := T#10S;
   T38.IN := FALSE;
   T39.PT := T#0MS;
   T39.IN := FALSE;
   T40.PT := T#0MS;
   T40.IN := FALSE;
   T41.PT := T#650MS;
   T41.IN := FALSE;
   T42.PT := T#3S;
   T42.IN := FALSE;
   T43.PT := T#0MS;
   T43.IN := FALSE;
   T44.PT := T#3S_500MS;
   T44.IN := FALSE;
   T45.PT := T#1S;
   T45.IN := FALSE;
   T46.PT := T#0MS;
   T46.IN := FALSE;
   T47.PT := T#500MS;
   T47.IN := TRUE;
   T48.PT := T#0MS;
   T48.IN := FALSE;
   T49.PT := T#0MS;
   T49.IN := FALSE;
   T50.PT := T#0MS;
   T50.IN := FALSE;
   T51.PT := T#4S;
   T51.IN := TRUE;
   T52.PT := T#0MS;
   T52.IN := FALSE;
   T53.PT := T#0MS;
   T53.IN := TRUE;
   T54.PT := T#0MS;
   T54.IN := FALSE;
   T55.PT := T#0MS;
   T55.IN := FALSE;
   T56.PT := T#0MS;
   T56.IN := FALSE;
   T57.PT := T#0MS;
   T57.IN := FALSE;
   T58.PT := T#0MS;
   T58.IN := FALSE;
   T59.PT := T#0MS;
   T59.IN := FALSE;
   T60.PT := T#0MS;
   T60.IN := FALSE;
   T61.PT := T#0MS;
   T61.IN := FALSE;
   T62.PT := T#0MS;
   T62.IN := FALSE;
   T63.PT := T#0MS;
   T63.IN := FALSE;
   T64.PT := T#0MS;
   T64.IN := FALSE;
   T65.PT := T#0MS;
   T65.IN := FALSE;
   T66.PT := T#0MS;
   T66.IN := FALSE;
   T67.PT := T#0MS;
   T67.IN := FALSE;
   T68.PT := T#0MS;
   T68.IN := FALSE;
   T69.PT := T#0MS;
   T69.IN := FALSE;
   T70.PT := T#0MS;
   T70.IN := FALSE;
   T71.PT := T#0MS;
   T71.IN := FALSE;
   T72.PT := T#0MS;
   T72.IN := FALSE;
   T73.PT := T#0MS;
   T73.IN := FALSE;
   T74.PT := T#0MS;
   T74.IN := FALSE;
   T75.PT := T#0MS;
   T75.IN := FALSE;
   T76.PT := T#0MS;
   T76.IN := FALSE;
   T77.PT := T#0MS;
   T77.IN := FALSE;
   T78.PT := T#0MS;
   T78.IN := FALSE;
   T79.PT := T#2S;
   T79.IN := FALSE;
   T80.PT := T#1S;
   T80.IN := TRUE;
   T81.PT := T#700MS;
   T81.IN := TRUE;
   T82.PT := T#10S;
   T82.IN := FALSE;
   T83.PT := T#500MS;
   T83.IN := FALSE;
   T84.PT := T#400MS;
   T84.IN := TRUE;
   T85.PT := T#0MS;
   T85.IN := FALSE;
   T86.PT := T#300MS;
   T86.IN := FALSE;
   T87.PT := T#0MS;
   T87.IN := FALSE;
   T88.PT := T#0MS;
   T88.IN := FALSE;
   T89.PT := T#0MS;
   T89.IN := FALSE;
   T90.PT := T#2S;
   T90.IN := FALSE;
   T91.PT := T#1S;
   T91.IN := FALSE;
   T92.PT := T#0MS;
   T92.IN := FALSE;
   T93.PT := T#0MS;
   T93.IN := FALSE;
   T94.PT := T#0MS;
   T94.IN := FALSE;
   T95.PT := T#0MS;
   T95.IN := FALSE;
   T96.PT := T#0MS;
   T96.IN := FALSE;
   T97.PT := T#0MS;
   T97.IN := FALSE;
   T98.PT := T#0MS;
   T98.IN := FALSE;
   T99.PT := T#0MS;
   T99.IN := FALSE;
   T100.PT := T#0MS;
   T100.IN := FALSE;
   T101.PT := T#0MS;
   T101.IN := FALSE;
   T102.PT := T#0MS;
   T102.IN := FALSE;
   T103.PT := T#0MS;
   T103.IN := FALSE;
   T104.PT := T#0MS;
   T104.IN := FALSE;
   T105.PT := T#0MS;
   T105.IN := FALSE;
   T106.PT := T#0MS;
   T106.IN := FALSE;
   T107.PT := T#0MS;
   T107.IN := FALSE;
   T108.PT := T#0MS;
   T108.IN := FALSE;
   T109.PT := T#0MS;
   T109.IN := FALSE;
   T110.PT := T#0MS;
   T110.IN := FALSE;
   T111.PT := T#0MS;
   T111.IN := FALSE;
   T112.PT := T#0MS;
   T112.IN := FALSE;
   T113.PT := T#0MS;
   T113.IN := FALSE;
   T114.PT := T#0MS;
   T114.IN := FALSE;
   T115.PT := T#0MS;
   T115.IN := FALSE;
   T116.PT := T#0MS;
   T116.IN := FALSE;
   T117.PT := T#0MS;
   T117.IN := FALSE;
   T118.PT := T#0MS;
   T118.IN := FALSE;
   T119.PT := T#0MS;
   T119.IN := FALSE;
   T120.PT := T#0MS;
   T120.IN := FALSE;
   T121.PT := T#0MS;
   T121.IN := FALSE;
   T122.PT := T#0MS;
   T122.IN := FALSE;
   T123.PT := T#0MS;
   T123.IN := FALSE;
   T124.PT := T#0MS;
   T124.IN := FALSE;
   T125.PT := T#0MS;
   T125.IN := FALSE;
   T126.PT := T#0MS;
   T126.IN := FALSE;
   T127.PT := T#0MS;
   T127.IN := FALSE;
   T128.PT := T#0MS;
   T128.IN := FALSE;
   T129.PT := T#0MS;
   T129.IN := FALSE;
   T130.PT := T#0MS;
   T130.IN := FALSE;
   T131.PT := T#0MS;
   T131.IN := FALSE;
   T132.PT := T#3S;
   T132.IN := FALSE;
   T133.PT := T#0MS;
   T133.IN := FALSE;
   T134.PT := T#0MS;
   T134.IN := FALSE;
   T135.PT := T#1S_500MS;
   T135.IN := TRUE;
   T136.PT := T#0MS;
   T136.IN := FALSE;
   T137.PT := T#0MS;
   T137.IN := FALSE;
   T138.PT := T#0MS;
   T138.IN := FALSE;
   T139.PT := T#0MS;
   T139.IN := FALSE;
   T140.PT := T#0MS;
   T140.IN := FALSE;
   T141.PT := T#0MS;
   T141.IN := FALSE;
   T142.PT := T#0MS;
   T142.IN := FALSE;
   T143.PT := T#0MS;
   T143.IN := FALSE;
   T144.PT := T#0MS;
   T144.IN := FALSE;
   T145.PT := T#0MS;
   T145.IN := FALSE;
   T146.PT := T#0MS;
   T146.IN := FALSE;
   T147.PT := T#0MS;
   T147.IN := FALSE;
   T148.PT := T#0MS;
   T148.IN := FALSE;
   T149.PT := T#0MS;
   T149.IN := FALSE;
   T150.PT := T#0MS;
   T150.IN := FALSE;
   T151.PT := T#0MS;
   T151.IN := FALSE;
   T152.PT := T#0MS;
   T152.IN := FALSE;
   T153.PT := T#0MS;
   T153.IN := FALSE;
   T154.PT := T#0MS;
   T154.IN := FALSE;
   T155.PT := T#0MS;
   T155.IN := FALSE;
   T156.PT := T#0MS;
   T156.IN := FALSE;
   T157.PT := T#0MS;
   T157.IN := FALSE;
   T158.PT := T#0MS;
   T158.IN := FALSE;
   T159.PT := T#0MS;
   T159.IN := FALSE;
   T160.PT := T#0MS;
   T160.IN := FALSE;
   T161.PT := T#0MS;
   T161.IN := FALSE;
   T162.PT := T#0MS;
   T162.IN := FALSE;
   T163.PT := T#0MS;
   T163.IN := FALSE;
   T164.PT := T#0MS;
   T164.IN := FALSE;
   T165.PT := T#0MS;
   T165.IN := FALSE;
   T166.PT := T#0MS;
   T166.IN := FALSE;
   T167.PT := T#0MS;
   T167.IN := FALSE;
   T168.PT := T#0MS;
   T168.IN := FALSE;
   T169.PT := T#0MS;
   T169.IN := FALSE;
   T170.PT := T#0MS;
   T170.IN := FALSE;
   T171.PT := T#0MS;
   T171.IN := FALSE;
   T172.PT := T#0MS;
   T172.IN := FALSE;
   T173.PT := T#0MS;
   T173.IN := FALSE;
   T174.PT := T#0MS;
   T174.IN := FALSE;
   T175.PT := T#0MS;
   T175.IN := FALSE;
   T176.PT := T#0MS;
   T176.IN := FALSE;
   T177.PT := T#0MS;
   T177.IN := FALSE;
   T178.PT := T#0MS;
   T178.IN := FALSE;
   T179.PT := T#0MS;
   T179.IN := FALSE;
   T180.PT := T#0MS;
   T180.IN := FALSE;
   T181.PT := T#0MS;
   T181.IN := FALSE;
   T182.PT := T#0MS;
   T182.IN := FALSE;
   T183.PT := T#0MS;
   T183.IN := FALSE;
   T184.PT := T#0MS;
   T184.IN := FALSE;
   T185.PT := T#0MS;
   T185.IN := FALSE;
   T186.PT := T#0MS;
   T186.IN := FALSE;
   T187.PT := T#0MS;
   T187.IN := FALSE;
   T188.PT := T#0MS;
   T188.IN := FALSE;
   T189.PT := T#0MS;
   T189.IN := FALSE;
   T190.PT := T#0MS;
   T190.IN := FALSE;
   T191.PT := T#0MS;
   T191.IN := FALSE;
   T192.PT := T#0MS;
   T192.IN := FALSE;
   T193.PT := T#0MS;
   T193.IN := FALSE;
   T194.PT := T#0MS;
   T194.IN := FALSE;
   T195.PT := T#0MS;
   T195.IN := FALSE;
   T196.PT := T#0MS;
   T196.IN := FALSE;
   T197.PT := T#0MS;
   T197.IN := FALSE;
   T198.PT := T#0MS;
   T198.IN := FALSE;
   T199.PT := T#0MS;
   T199.IN := FALSE;
   T200.PT := T#5S;
   T200.IN := FALSE;
   T201.PT := T#200MS;
   T201.IN := TRUE;
   T202.PT := T#200MS;
   T202.IN := FALSE;
   T203.PT := T#1S;
   T203.IN := FALSE;
   T204.PT := T#0MS;
   T204.IN := FALSE;
   T205.PT := T#200MS;
   T205.IN := FALSE;
   T206.PT := T#200MS;
   T206.IN := FALSE;
   T207.PT := T#200MS;
   T207.IN := TRUE;
   T208.PT := T#0MS;
   T208.IN := FALSE;
   T209.PT := T#0MS;
   T209.IN := FALSE;
   T210.PT := T#200MS;
   T210.IN := FALSE;
   T211.PT := T#10S;
   T211.IN := FALSE;
   T212.PT := T#0MS;
   T212.IN := FALSE;
   T213.PT := T#3S;
   T213.IN := FALSE;
   T214.PT := T#1S_500MS;
   T214.IN := TRUE;
   T215.PT := T#2S;
   T215.IN := FALSE;
   T216.PT := T#5S;
   T216.IN := FALSE;
END_DATA_BLOCK

ORGANIZATION_BLOCK "Main"   // OB1, LAD, ProgramCycle
TITLE = "Main Program Sweep (Cycle)"
{ S7_Optimized_Access := 'TRUE' }
VERSION : 0.1
// stored: AutoNumber false, IsIECCheckEnabled false, SetENOAutomatically false
   VAR_TEMP
      SALDATORE : Bool;
      PORTA : Bool;
      ESAUR_FILM : Bool;
      STR_FASCIA : Bool;
      STR_CORDA : Bool;
      CONTRASTO : Bool;
      PRESSORE : Bool;
      PRESS_RECT : Bool;
      AUTO_CENTR : Bool;
      TOP : Bool;
      BRAKE : Bool;   // Table phase
      PHASE : Bool;   // Table brake
   END_VAR
   VAR_TEMP   // added for the SCL form of the ladder/FBD networks
      _w1 : Bool;
      _w2 : Bool;
      _w3 : Bool;
   END_VAR
BEGIN

REGION Network 1: Bit always on
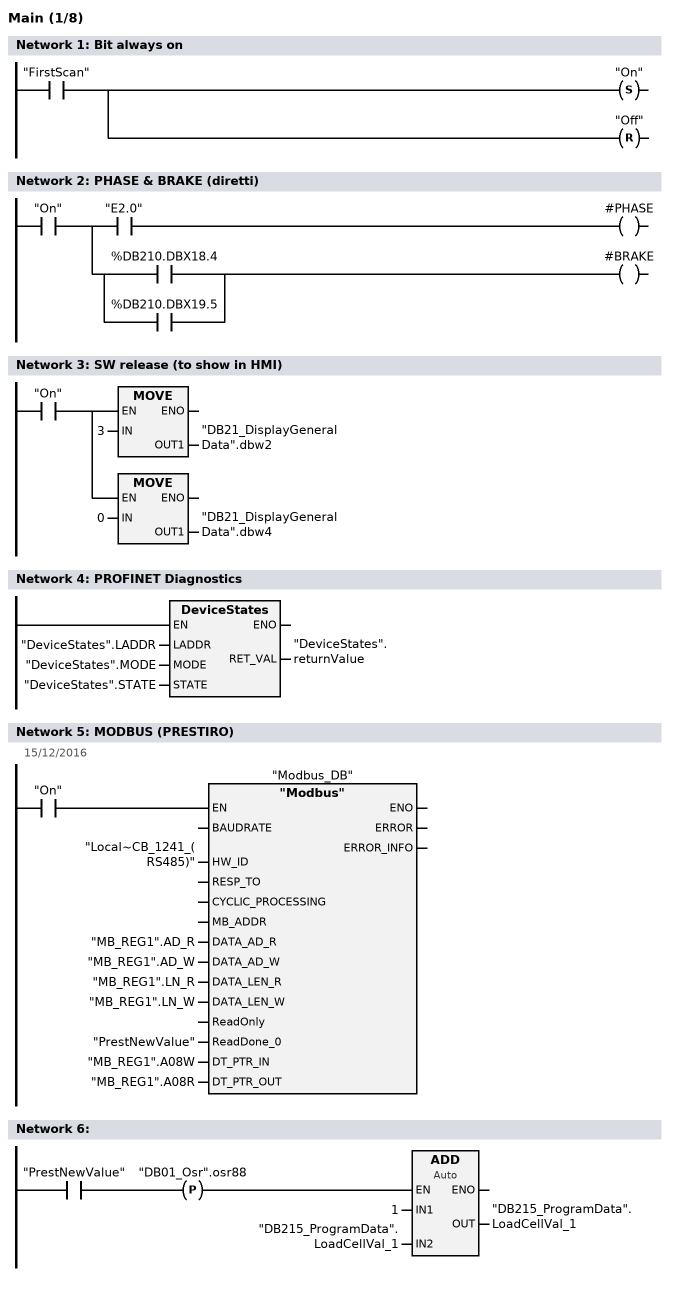
   RUNG wire#powerrail
      Contact( "FirstScan" )
      wire#w1
      S_Coil( "On" )
   END_RUNG
   RUNG wire#w1
      R_Coil( "Off" )
   END_RUNG
   // the same network as SCL:
   IF "FirstScan" THEN
       "On" := TRUE;
       "Off" := FALSE;
   END_IF;
END_REGION

REGION Network 2: PHASE & BRAKE (diretti)
   RUNG wire#powerrail
      Contact( "On" )
      wire#w1
      Contact( "E2.0" )
      Coil( #PHASE )
   END_RUNG
   RUNG wire#w1
      Contact( %DB210.DBX18.4 )
      wire#w2
      Coil( #BRAKE )
   END_RUNG
   RUNG wire#w1
      Contact( %DB210.DBX19.5 )
   END_RUNG wire#w2
   // the same network as SCL:
   #PHASE := "On" AND "E2.0";
   #BRAKE := "On" AND (%DB210.DBX18.4 OR %DB210.DBX19.5);
END_REGION

REGION Network 3: SW release (to show in HMI)
   RUNG wire#powerrail
      Contact( "On" )
      wire#w1
      Move(in := 3, out1 => "DB21_DisplayGeneralData".dbw2)
   END_RUNG
   RUNG wire#w1
      Move(in := 0, out1 => "DB21_DisplayGeneralData".dbw4)
   END_RUNG
   // the same network as SCL:
   IF "On" THEN
       "DB21_DisplayGeneralData".dbw2 := 3;
       "DB21_DisplayGeneralData".dbw4 := 0;
   END_IF;
END_REGION

REGION Network 4: PROFINET Diagnostics
   RUNG wire#powerrail
      DeviceStates(LADDR := "DeviceStates".LADDR, MODE := "DeviceStates".MODE, STATE := "DeviceStates".STATE, Ret_Val => "DeviceStates".returnValue)
   END_RUNG
   // the same network as SCL:
   "DeviceStates".returnValue := DeviceStates(LADDR := "DeviceStates".LADDR,
                           MODE := "DeviceStates".MODE,
                           STATE := "DeviceStates".STATE);
END_REGION

REGION Network 5: MODBUS (PRESTIRO)
   // 15/12/2016
   RUNG wire#powerrail
      Contact( "On" )
      "Modbus_DB"(BAUDRATE :=, HW_ID := "Local~CB_1241_(RS485)", RESP_TO :=, CYCLIC_PROCESSING :=, MB_ADDR :=, DATA_AD_R := "MB_REG1".AD_R, DATA_AD_W := "MB_REG1".AD_W, DATA_LEN_R := "MB_REG1".LN_R, DATA_LEN_W := "MB_REG1".LN_W, ReadOnly :=, ReadDone_0 := "PrestNewValue", DT_PTR_IN := "MB_REG1".A08W, DT_PTR_OUT := "MB_REG1".A08R, ERROR =>, ERROR_INFO =>)
   END_RUNG
   // the same network as SCL:
   IF "On" THEN
       "Modbus_DB"(HW_ID := "Local~CB_1241_(RS485)",   // "Modbus"
                   DATA_AD_R := "MB_REG1".AD_R,
                   DATA_AD_W := "MB_REG1".AD_W,
                   DATA_LEN_R := "MB_REG1".LN_R,
                   DATA_LEN_W := "MB_REG1".LN_W,
                   ReadDone_0 := "PrestNewValue",
                   DT_PTR_IN := "MB_REG1".A08W,
                   DT_PTR_OUT := "MB_REG1".A08R);
   END_IF;
END_REGION

REGION Network 6
   RUNG wire#powerrail
      Contact( "PrestNewValue" )
      P_Trig( "DB01_Osr".osr88 )
      Add(in1 := 1, in2 := "DB215_ProgramData".LoadCellVal_1, out => "DB215_ProgramData".LoadCellVal_1)
   END_RUNG
   // the same network as SCL:
   #_w1 := "PrestNewValue" AND NOT "DB01_Osr".osr88;   // rising edge
   "DB01_Osr".osr88 := "PrestNewValue";
   IF #_w1 THEN "DB215_ProgramData".LoadCellVal_1 := 1 + "DB215_ProgramData".LoadCellVal_1; END_IF;
END_REGION

REGION Network 7: Reset Modbus errors
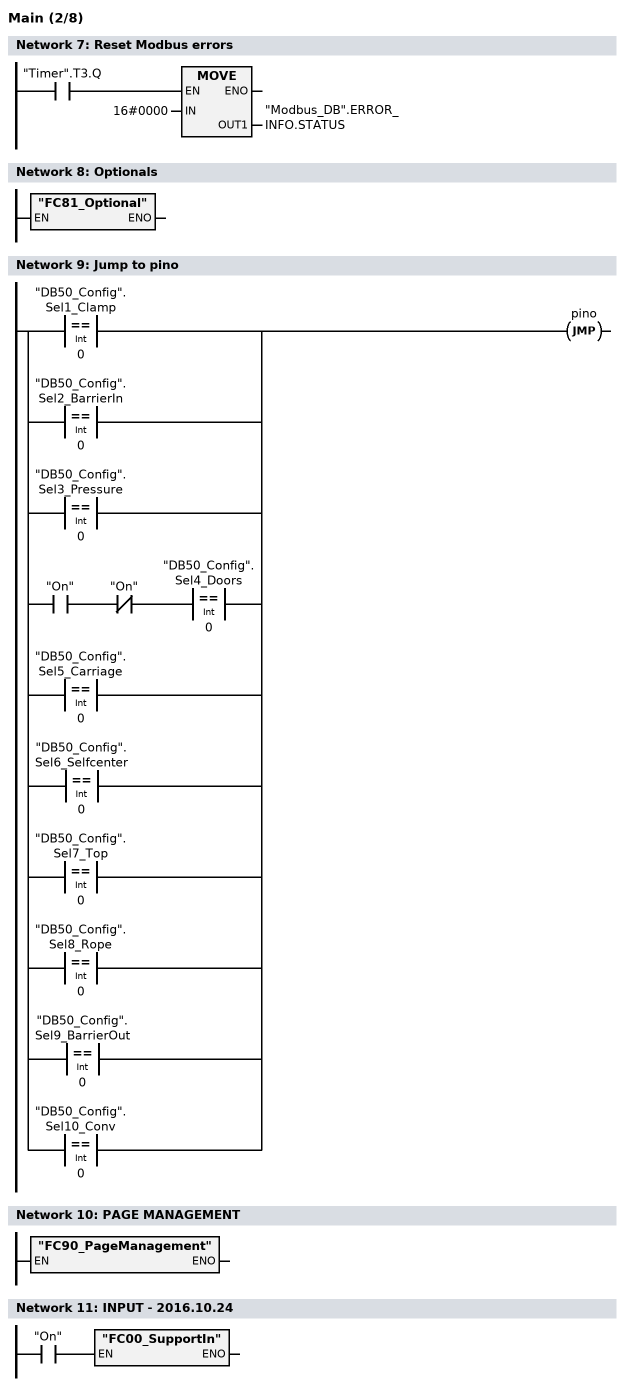
   RUNG wire#powerrail
      Contact( "Timer".T3.Q )
      Move(in := 16#0000, out1 => "Modbus_DB".ERROR_INFO.STATUS)
   END_RUNG
   // the same network as SCL:
   IF "Timer".T3.Q THEN "Modbus_DB".ERROR_INFO.STATUS := 16#0000; END_IF;
END_REGION

REGION Network 8: Optionals
   RUNG wire#powerrail
      "FC81_Optional"()
   END_RUNG
   // the same network as SCL:
   "FC81_Optional"();
END_REGION

REGION Network 9: Jump to pino
   RUNG wire#powerrail
      { S7_Templates := "SrcType := Int" } EQ_Contact(in1 := "DB50_Config".Sel1_Clamp, in2 := 0)
      wire#w1
      JumpCoil( pino )
   END_RUNG
   RUNG wire#powerrail
      { S7_Templates := "SrcType := Int" } EQ_Contact(in1 := "DB50_Config".Sel2_BarrierIn, in2 := 0)
   END_RUNG wire#w1
   RUNG wire#powerrail
      { S7_Templates := "SrcType := Int" } EQ_Contact(in1 := "DB50_Config".Sel3_Pressure, in2 := 0)
   END_RUNG wire#w1
   RUNG wire#powerrail
      Contact( "On" )
      I_Contact( "On" )
      { S7_Templates := "SrcType := Int" } EQ_Contact(in1 := "DB50_Config".Sel4_Doors, in2 := 0)
   END_RUNG wire#w1
   RUNG wire#powerrail
      { S7_Templates := "SrcType := Int" } EQ_Contact(in1 := "DB50_Config".Sel5_Carriage, in2 := 0)
   END_RUNG wire#w1
   RUNG wire#powerrail
      { S7_Templates := "SrcType := Int" } EQ_Contact(in1 := "DB50_Config".Sel6_Selfcenter, in2 := 0)
   END_RUNG wire#w1
   RUNG wire#powerrail
      { S7_Templates := "SrcType := Int" } EQ_Contact(in1 := "DB50_Config".Sel7_Top, in2 := 0)
   END_RUNG wire#w1
   RUNG wire#powerrail
      { S7_Templates := "SrcType := Int" } EQ_Contact(in1 := "DB50_Config".Sel8_Rope, in2 := 0)
   END_RUNG wire#w1
   RUNG wire#powerrail
      { S7_Templates := "SrcType := Int" } EQ_Contact(in1 := "DB50_Config".Sel9_BarrierOut, in2 := 0)
   END_RUNG wire#w1
   RUNG wire#powerrail
      { S7_Templates := "SrcType := Int" } EQ_Contact(in1 := "DB50_Config".Sel10_Conv, in2 := 0)
   END_RUNG wire#w1
   // the same network as SCL:
   IF ("DB50_Config".Sel1_Clamp = 0) OR ("DB50_Config".Sel2_BarrierIn = 0) OR ("DB50_Config".Sel3_Pressure = 0) OR ("On" AND NOT "On" AND ("DB50_Config".Sel4_Doors = 0)) OR ("DB50_Config".Sel5_Carriage = 0) OR ("DB50_Config".Sel6_Selfcenter = 0) OR ("DB50_Config".Sel7_Top = 0) OR ("DB50_Config".Sel8_Rope = 0) OR ("DB50_Config".Sel9_BarrierOut = 0) OR ("DB50_Config".Sel10_Conv = 0) THEN
       GOTO pino;
   END_IF;
END_REGION

REGION Network 10: PAGE MANAGEMENT
   RUNG wire#powerrail
      "FC90_PageManagement"()
   END_RUNG
   // the same network as SCL:
   "FC90_PageManagement"();
END_REGION

REGION Network 11: INPUT - 2016.10.24
   RUNG wire#powerrail
      Contact( "On" )
      "FC00_SupportIn"()
   END_RUNG
   // the same network as SCL:
   IF "On" THEN "FC00_SupportIn"(); END_IF;
END_REGION

REGION Network 12: ACCESSORIES (CONFIGURATION)
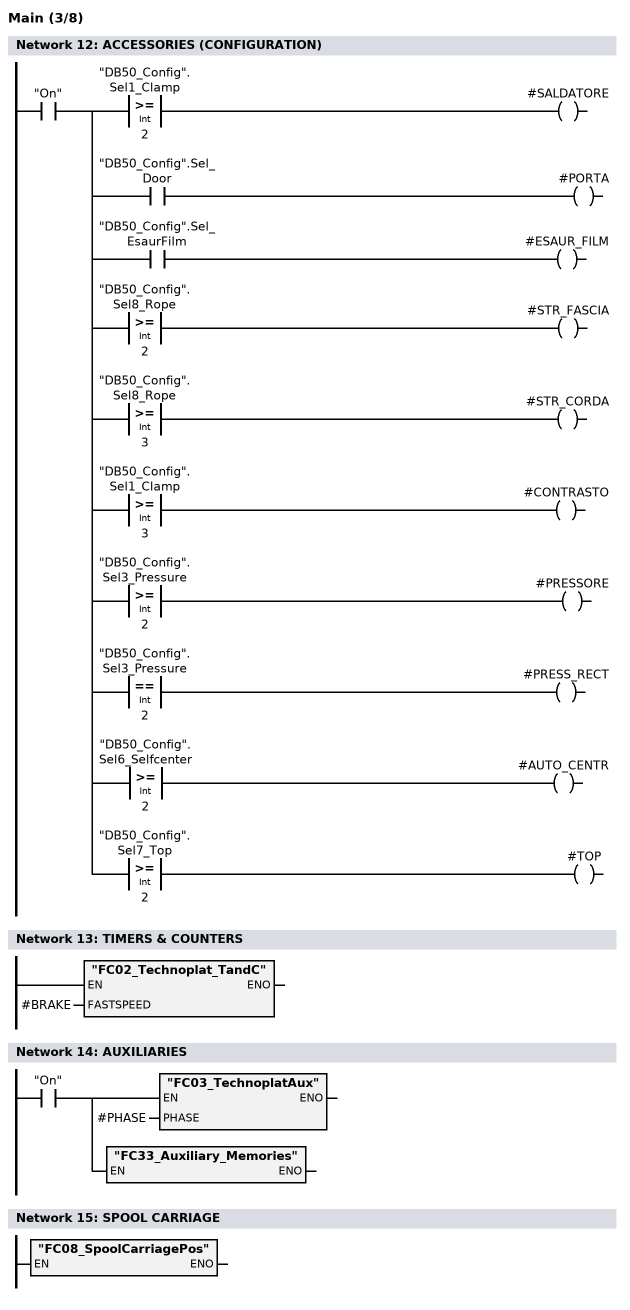
   RUNG wire#powerrail
      Contact( "On" )
      wire#w1
      { S7_Templates := "SrcType := Int" } GE_Contact(in1 := "DB50_Config".Sel1_Clamp, in2 := 2)
      Coil( #SALDATORE )
   END_RUNG
   RUNG wire#w1
      Contact( "DB50_Config".Sel_Door )
      Coil( #PORTA )
   END_RUNG
   RUNG wire#w1
      Contact( "DB50_Config".Sel_EsaurFilm )
      Coil( #ESAUR_FILM )
   END_RUNG
   RUNG wire#w1
      { S7_Templates := "SrcType := Int" } GE_Contact(in1 := "DB50_Config".Sel8_Rope, in2 := 2)
      Coil( #STR_FASCIA )
   END_RUNG
   RUNG wire#w1
      { S7_Templates := "SrcType := Int" } GE_Contact(in1 := "DB50_Config".Sel8_Rope, in2 := 3)
      Coil( #STR_CORDA )
   END_RUNG
   RUNG wire#w1
      { S7_Templates := "SrcType := Int" } GE_Contact(in1 := "DB50_Config".Sel1_Clamp, in2 := 3)
      Coil( #CONTRASTO )
   END_RUNG
   RUNG wire#w1
      { S7_Templates := "SrcType := Int" } GE_Contact(in1 := "DB50_Config".Sel3_Pressure, in2 := 2)
      Coil( #PRESSORE )
   END_RUNG
   RUNG wire#w1
      { S7_Templates := "SrcType := Int" } EQ_Contact(in1 := "DB50_Config".Sel3_Pressure, in2 := 2)
      Coil( #PRESS_RECT )
   END_RUNG
   RUNG wire#w1
      { S7_Templates := "SrcType := Int" } GE_Contact(in1 := "DB50_Config".Sel6_Selfcenter, in2 := 2)
      Coil( #AUTO_CENTR )
   END_RUNG
   RUNG wire#w1
      { S7_Templates := "SrcType := Int" } GE_Contact(in1 := "DB50_Config".Sel7_Top, in2 := 2)
      Coil( #TOP )
   END_RUNG
   // the same network as SCL:
   #SALDATORE := "On" AND ("DB50_Config".Sel1_Clamp >= 2);
   #PORTA := "On" AND "DB50_Config".Sel_Door;
   #ESAUR_FILM := "On" AND "DB50_Config".Sel_EsaurFilm;
   #STR_FASCIA := "On" AND ("DB50_Config".Sel8_Rope >= 2);
   #STR_CORDA := "On" AND ("DB50_Config".Sel8_Rope >= 3);
   #CONTRASTO := "On" AND ("DB50_Config".Sel1_Clamp >= 3);
   #PRESSORE := "On" AND ("DB50_Config".Sel3_Pressure >= 2);
   #PRESS_RECT := "On" AND ("DB50_Config".Sel3_Pressure = 2);
   #AUTO_CENTR := "On" AND ("DB50_Config".Sel6_Selfcenter >= 2);
   #TOP := "On" AND ("DB50_Config".Sel7_Top >= 2);
END_REGION

REGION Network 13: TIMERS & COUNTERS
   RUNG wire#powerrail
      "FC02_Technoplat_TandC"(FASTSPEED := #BRAKE)
   END_RUNG
   // the same network as SCL:
   "FC02_Technoplat_TandC"(FASTSPEED := #BRAKE);
END_REGION

REGION Network 14: AUXILIARIES
   RUNG wire#powerrail
      Contact( "On" )
      wire#w1
      "FC03_TechnoplatAux"(PHASE := #PHASE)
   END_RUNG
   RUNG wire#w1
      "FC33_Auxiliary_Memories"()
   END_RUNG
   // the same network as SCL:
   #_w1 := "On";
   IF #_w1 THEN
       "FC03_TechnoplatAux"(PHASE := #PHASE);
       "FC33_Auxiliary_Memories"();
   END_IF;
END_REGION

REGION Network 15: SPOOL CARRIAGE
   RUNG wire#powerrail
      "FC08_SpoolCarriagePos"()
   END_RUNG
   // the same network as SCL:
   "FC08_SpoolCarriagePos"();
END_REGION

REGION Network 16: ROTATION TABLE
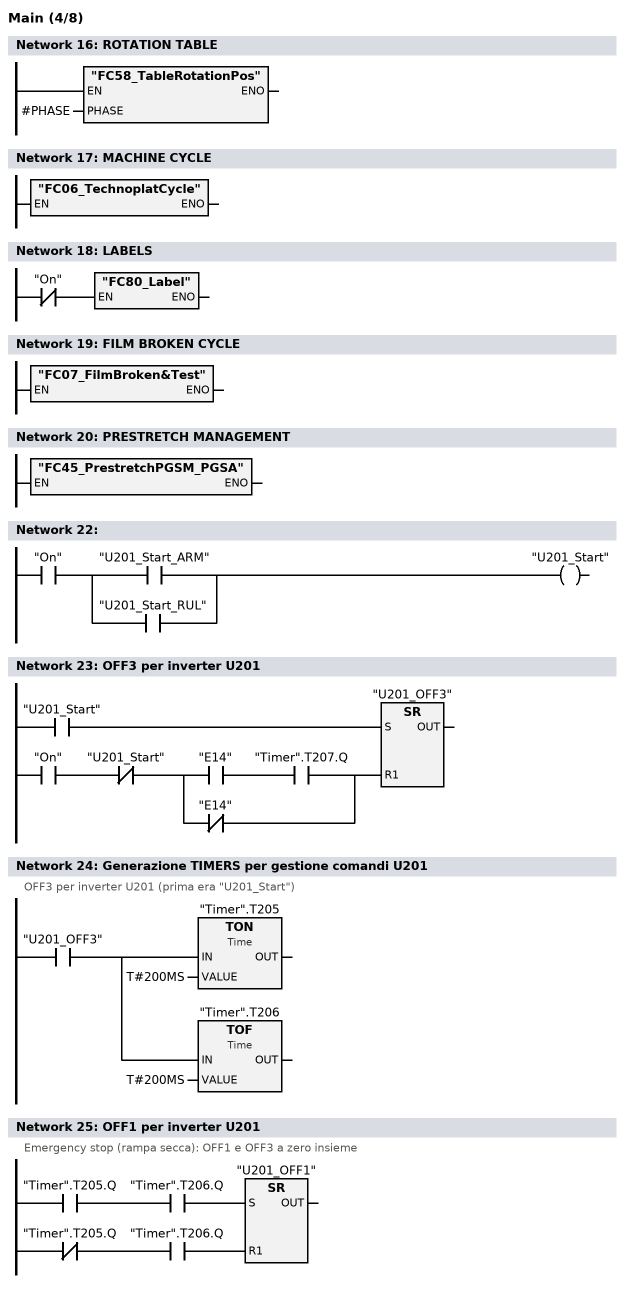
   RUNG wire#powerrail
      "FC58_TableRotationPos"(PHASE := #PHASE)
   END_RUNG
   // the same network as SCL:
   "FC58_TableRotationPos"(PHASE := #PHASE);
END_REGION

REGION Network 17: MACHINE CYCLE
   RUNG wire#powerrail
      "FC06_TechnoplatCycle"()
   END_RUNG
   // the same network as SCL:
   "FC06_TechnoplatCycle"();
END_REGION

REGION Network 18: LABELS
   RUNG wire#powerrail
      I_Contact( "On" )
      "FC80_Label"()
   END_RUNG
   // the same network as SCL:
   IF NOT "On" THEN "FC80_Label"(); END_IF;
END_REGION

REGION Network 19: FILM BROKEN CYCLE
   RUNG wire#powerrail
      "FC07_FilmBroken&Test"()
   END_RUNG
   // the same network as SCL:
   "FC07_FilmBroken&Test"();
END_REGION

REGION Network 20: PRESTRETCH MANAGEMENT
   RUNG wire#powerrail
      "FC45_PrestretchPGSM_PGSA"()
   END_RUNG
   // the same network as SCL:
   "FC45_PrestretchPGSM_PGSA"();
END_REGION

REGION Network 21: - - - GESTIONE INVERTER PROFINET - - -
END_REGION

REGION Network 22
   RUNG wire#powerrail
      Contact( "On" )
      wire#w1
      Contact( "U201_Start_ARM" )
      wire#w2
      Coil( "U201_Start" )
   END_RUNG
   RUNG wire#w1
      Contact( "U201_Start_RUL" )
   END_RUNG wire#w2
   // the same network as SCL:
   "U201_Start" := "On" AND ("U201_Start_ARM" OR "U201_Start_RUL");
END_REGION

REGION Network 23: OFF3 per inverter U201
   RUNG wire#powerrail
      Contact( "U201_Start" )
      S_SR(operand := "U201_OFF3", r1 := wire#w2)
   END_RUNG
   RUNG wire#powerrail
      Contact( "On" )
      I_Contact( "U201_Start" )
      wire#w1
      Contact( "E14" )
      Contact( "Timer".T207.Q )
   END_RUNG wire#w2
   RUNG wire#w1
      I_Contact( "E14" )
   END_RUNG wire#w2
   // the same network as SCL:
   IF "U201_Start" THEN
       "U201_OFF3" := TRUE;   // SR flip-flop
   END_IF;
   IF "On" AND NOT "U201_Start" AND (("E14" AND "Timer".T207.Q) OR NOT "E14") THEN
       "U201_OFF3" := FALSE;
   END_IF;
END_REGION

REGION Network 24: Generazione TIMERS per gestione comandi U201
   // OFF3 per inverter U201 (prima era "U201_Start")
   "Timer".T205.TON(IN := "U201_OFF3", PT := T#200MS);   // TON coil
   "Timer".T206.TOF(IN := "U201_OFF3", PT := T#200MS);   // TOF coil
END_REGION

REGION Network 25: OFF1 per inverter U201
   // Emergency stop (rampa secca): OFF1 e OFF3 a zero insieme
   RUNG wire#powerrail
      Contact( "Timer".T205.Q )
      Contact( "Timer".T206.Q )
      S_SR(operand := "U201_OFF1", r1 := wire#w1)
   END_RUNG
   RUNG wire#powerrail
      I_Contact( "Timer".T205.Q )
      Contact( "Timer".T206.Q )
   END_RUNG wire#w1
   // the same network as SCL:
   IF "Timer".T205.Q AND "Timer".T206.Q THEN
       "U201_OFF1" := TRUE;   // SR flip-flop
   END_IF;
   IF NOT "Timer".T205.Q AND "Timer".T206.Q THEN "U201_OFF1" := FALSE; END_IF;
END_REGION

